# B&R Automation Studio project NAINV104C00R8L515F00 (part 33)

#### Act_Background_SendBoardDepartedLane3.st - Do Not Change!!!
```iecst
(** 2021-08-01 **)
ACTION Act_Background_SendBoardDepartedLane3: //Send after our machine send out "TransportFinished" message to downstream

	IF eStatus2 <> Error THEN
		IF tySServiceDescriptionRcv.tyData.tySupportedFeatures.bFeatureBoardTracking = TRUE AND p_tyParam.bFeatureBoardTracking AND bHandshakeDone THEN
			IF EDGEPOS(p_bDSHermesTransportFinished3) THEN

				fHermesAddOneMsgSend(ADR(a_eMsgSend) , ADR(udiMsgSendBffr) , HermesMsgTypeBoardDeparted3);

				tyBoardDeparted3.tyData.sMachineId     	        := p_sMcId;
			    tyBoardDeparted3.tyData.iDownstreamLaneId    	:= p_tyHermesConfiguration.a_tyDSParam[2].iLaneID;
			    tyBoardDeparted3.tyData.sDownstreamInterfaceId  := p_tyHermesConfiguration.a_tyDSParam[2].sDownstreamInterfaceId;
                tyBoardDeparted3.tyData.sMagazineId           	:= sMagazineId;
		    	tyBoardDeparted3.tyData.iSlotId     	        := iSlotId;
		    	tyBoardDeparted3.tyData.eBoadTransfer    	    := p_eBoardTransfer3;
	            tyBoardDeparted3.tyData.sBoardId     	        := p_tyDSBoardDeparted3.tyData.sBoardId;
		    	tyBoardDeparted3.tyData.sBoardIdCreatedBy     	:= p_tyDSBoardDeparted3.tyData.sBoardIdCreatedBy;
		    	tyBoardDeparted3.tyData.eFailedBoard			:= p_tyDSBoardDeparted3.tyData.eFailedBoard;
				tyBoardDeparted3.tyData.sProductTypeId			:= p_tyDSBoardDeparted3.tyData.sProductTypeId;
				tyBoardDeparted3.tyData.eFlippedBoard			:= p_tyDSBoardDeparted3.tyData.eFlippedBoard;
				tyBoardDeparted3.tyData.sTopBarcode				:= p_tyDSBoardDeparted3.tyData.sTopBarcode;
				tyBoardDeparted3.tyData.sBottomBarcode			:= p_tyDSBoardDeparted3.tyData.sBottomBarcode;
				tyBoardDeparted3.tyData.rLength					:= p_tyDSBoardDeparted3.tyData.rLength;
				tyBoardDeparted3.tyData.rWidth				    := p_tyDSBoardDeparted3.tyData.rWidth;
				tyBoardDeparted3.tyData.rThickness				:= p_tyDSBoardDeparted3.tyData.rThickness;
				tyBoardDeparted3.tyData.rConveyorSpeed		    := p_tyDSBoardDeparted3.tyData.rConveyorSpeed;
				tyBoardDeparted3.tyData.rTopClearanceHeight		:= p_tyDSBoardDeparted3.tyData.rTopClearanceHeight;
				tyBoardDeparted3.tyData.rBottomClearanceHeight	:= p_tyDSBoardDeparted3.tyData.rBottomClearanceHeight;
				tyBoardDeparted3.tyData.rWeight					:= p_tyDSBoardDeparted3.tyData.rWeight;
				tyBoardDeparted3.tyData.sWorkOrdedId            := p_tyDSBoardDeparted3.tyData.sWorkOrderId;
				tyBoardDeparted3.tyData.sBatchId                := p_tyDSBoardDeparted3.tyData.sBatchId;

			    tyBoardDeparted3.tyAvl.bMachineId				:= tyBoardDeparted3.tyData.sMachineId <> '';
		     	tyBoardDeparted3.tyAvl.bDownstreamLaneId		:= tyBoardDeparted3.tyData.iDownstreamLaneId <> 0;
		    	tyBoardDeparted3.tyAvl.bDownstreamInterfaceId	:= tyBoardDeparted3.tyData.sDownstreamInterfaceId <> '';
		    	tyBoardDeparted3.tyAvl.bMagazineId		    	:= tyBoardDeparted3.tyData.sMagazineId <> '';
		    	tyBoardDeparted3.tyAvl.bSlotId				    := tyBoardDeparted3.tyData.iSlotId <> 0;
		    	tyBoardDeparted3.tyAvl.bBoardTransfer		    := TRUE;
				tyBoardDeparted3.tyAvl.bBoardId					:= tyBoardDeparted3.tyData.sBoardId <> '';
				tyBoardDeparted3.tyAvl.bBoardIdCreatedBy		:= tyBoardDeparted3.tyData.sBoardIdCreatedBy <> '';
				tyBoardDeparted3.tyAvl.bFailedBoard				:= TRUE;
				tyBoardDeparted3.tyAvl.bProductTypeId		   	:= tyBoardDeparted3.tyData.sProductTypeId <> '';
				tyBoardDeparted3.tyAvl.bFlippedBoard			:= TRUE;
				tyBoardDeparted3.tyAvl.bTopBarcode			    := tyBoardDeparted3.tyData.sTopBarcode <> '';
				tyBoardDeparted3.tyAvl.bBottomBarcode		    := tyBoardDeparted3.tyData.sBottomBarcode <> '';
				tyBoardDeparted3.tyAvl.bLength				    := tyBoardDeparted3.tyData.rLength <> 0;
				tyBoardDeparted3.tyAvl.bWidth				    := (tyBoardDeparted3.tyData.rWidth <> 0);
				tyBoardDeparted3.tyAvl.bThickness			    := (tyBoardDeparted3.tyData.rThickness <> 0);
				tyBoardDeparted3.tyAvl.bConveyorSpeed		    := tyBoardDeparted3.tyData.rConveyorSpeed <> 0;
				tyBoardDeparted3.tyAvl.bTopClearanceHeight	    := (tyBoardDeparted3.tyData.rTopClearanceHeight <> 0);
				tyBoardDeparted3.tyAvl.bBottomClearanceHeight	:= (tyBoardDeparted3.tyData.rBottomClearanceHeight <> 0);
		    	tyBoardDeparted3.tyAvl.bWeight				    := tyBoardDeparted3.tyData.rWeight <> 0;
				tyBoardDeparted3.tyAvl.bWorkOrderId				:= tyBoardDeparted3.tyData.sWorkOrdedId <> '';
				tyBoardDeparted3.tyAvl.bBatchId			    	:= tyBoardDeparted3.tyData.sBatchId <> '';

			END_IF

		END_IF

	END_IF

END_ACTION
```

#### Act_Background_SendBoardDepartedLane4.st - Do Not Change!!!
```iecst
(** 2021-08-01 **)
ACTION Act_Background_SendBoardDepartedLane4: //Send after our machine send out "TransportFinished" message to downstream

	IF eStatus2 <> Error THEN
		IF tySServiceDescriptionRcv.tyData.tySupportedFeatures.bFeatureBoardTracking = TRUE AND p_tyParam.bFeatureBoardTracking AND bHandshakeDone THEN
			IF EDGEPOS(p_bDSHermesTransportFinished4) THEN

				fHermesAddOneMsgSend(ADR(a_eMsgSend) , ADR(udiMsgSendBffr) , HermesMsgTypeBoardDeparted4);

				tyBoardDeparted4.tyData.sMachineId     	        := p_sMcId;
			    tyBoardDeparted4.tyData.iDownstreamLaneId    	:= p_tyHermesConfiguration.a_tyDSParam[3].iLaneID;
			    tyBoardDeparted4.tyData.sDownstreamInterfaceId  := p_tyHermesConfiguration.a_tyDSParam[3].sDownstreamInterfaceId;
                tyBoardDeparted4.tyData.sMagazineId           	:= sMagazineId;
		    	tyBoardDeparted4.tyData.iSlotId     	        := iSlotId;
		    	tyBoardDeparted4.tyData.eBoadTransfer    	    := p_eBoardTransfer4;
	            tyBoardDeparted4.tyData.sBoardId     	        := p_tyDSBoardDeparted4.tyData.sBoardId;
		    	tyBoardDeparted4.tyData.sBoardIdCreatedBy     	:= p_tyDSBoardDeparted4.tyData.sBoardIdCreatedBy;
		    	tyBoardDeparted4.tyData.eFailedBoard			:= p_tyDSBoardDeparted4.tyData.eFailedBoard;
				tyBoardDeparted4.tyData.sProductTypeId			:= p_tyDSBoardDeparted4.tyData.sProductTypeId;
				tyBoardDeparted4.tyData.eFlippedBoard			:= p_tyDSBoardDeparted4.tyData.eFlippedBoard;
				tyBoardDeparted4.tyData.sTopBarcode				:= p_tyDSBoardDeparted4.tyData.sTopBarcode;
				tyBoardDeparted4.tyData.sBottomBarcode			:= p_tyDSBoardDeparted4.tyData.sBottomBarcode;
				tyBoardDeparted4.tyData.rLength					:= p_tyDSBoardDeparted4.tyData.rLength;
				tyBoardDeparted4.tyData.rWidth				    := p_tyDSBoardDeparted4.tyData.rWidth;
				tyBoardDeparted4.tyData.rThickness				:= p_tyDSBoardDeparted4.tyData.rThickness;
				tyBoardDeparted4.tyData.rConveyorSpeed		    := p_tyDSBoardDeparted4.tyData.rConveyorSpeed;
				tyBoardDeparted4.tyData.rTopClearanceHeight		:= p_tyDSBoardDeparted4.tyData.rTopClearanceHeight;
				tyBoardDeparted4.tyData.rBottomClearanceHeight	:= p_tyDSBoardDeparted4.tyData.rBottomClearanceHeight;
				tyBoardDeparted4.tyData.rWeight					:= p_tyDSBoardDeparted4.tyData.rWeight;
				tyBoardDeparted4.tyData.sWorkOrdedId            := p_tyDSBoardDeparted4.tyData.sWorkOrderId;
				tyBoardDeparted4.tyData.sBatchId                := p_tyDSBoardDeparted4.tyData.sBatchId;

			    tyBoardDeparted4.tyAvl.bMachineId				:= tyBoardDeparted4.tyData.sMachineId <> '';
		     	tyBoardDeparted4.tyAvl.bDownstreamLaneId		:= tyBoardDeparted4.tyData.iDownstreamLaneId <> 0;
		    	tyBoardDeparted4.tyAvl.bDownstreamInterfaceId	:= tyBoardDeparted4.tyData.sDownstreamInterfaceId <> '';
		    	tyBoardDeparted4.tyAvl.bMagazineId		    	:= tyBoardDeparted4.tyData.sMagazineId <> '';
		    	tyBoardDeparted4.tyAvl.bSlotId				    := tyBoardDeparted4.tyData.iSlotId <> 0;
		    	tyBoardDeparted4.tyAvl.bBoardTransfer		    := TRUE;
				tyBoardDeparted4.tyAvl.bBoardId					:= tyBoardDeparted4.tyData.sBoardId <> '';
				tyBoardDeparted4.tyAvl.bBoardIdCreatedBy		:= tyBoardDeparted4.tyData.sBoardIdCreatedBy <> '';
				tyBoardDeparted4.tyAvl.bFailedBoard				:= TRUE;
				tyBoardDeparted4.tyAvl.bProductTypeId		   	:= tyBoardDeparted4.tyData.sProductTypeId <> '';
				tyBoardDeparted4.tyAvl.bFlippedBoard			:= TRUE;
				tyBoardDeparted4.tyAvl.bTopBarcode			    := tyBoardDeparted4.tyData.sTopBarcode <> '';
				tyBoardDeparted4.tyAvl.bBottomBarcode		    := tyBoardDeparted4.tyData.sBottomBarcode <> '';
				tyBoardDeparted4.tyAvl.bLength				    := tyBoardDeparted4.tyData.rLength <> 0;
				tyBoardDeparted4.tyAvl.bWidth				    := (tyBoardDeparted4.tyData.rWidth <> 0);
				tyBoardDeparted4.tyAvl.bThickness			    := (tyBoardDeparted4.tyData.rThickness <> 0);
				tyBoardDeparted4.tyAvl.bConveyorSpeed		    := tyBoardDeparted4.tyData.rConveyorSpeed <> 0;
				tyBoardDeparted4.tyAvl.bTopClearanceHeight	    := (tyBoardDeparted4.tyData.rTopClearanceHeight <> 0);
				tyBoardDeparted4.tyAvl.bBottomClearanceHeight	:= (tyBoardDeparted4.tyData.rBottomClearanceHeight <> 0);
		    	tyBoardDeparted4.tyAvl.bWeight				    := tyBoardDeparted4.tyData.rWeight <> 0;
				tyBoardDeparted4.tyAvl.bWorkOrderId				:= tyBoardDeparted4.tyData.sWorkOrdedId <> '';
				tyBoardDeparted4.tyAvl.bBatchId			    	:= tyBoardDeparted4.tyData.sBatchId <> '';

			END_IF

		END_IF

	END_IF

END_ACTION
```

#### Act_Background_TCPSend.st - Do Not Change!!!
```iecst
(** 2021-08-01 **)
ACTION Act_Background_TCPSend:

	//Message Send (Generate XML Message)
	IF a_eMsgSend[0] <> HermesMsgTypeNA THEN

		IF a_eMsgSend[0] = HermesMsgTypeCheckAlive THEN
			fHermesFormCheckAlive(ADR(a_tyXMLTableDataSnd) , p_tyDTStructure , tyCheckAliveSnd);
			fTableConvertToXML(ADR(sSnd) , ADR(udiSndMsgLen) , SIZEOF(sSnd) , ADR(a_tyXMLTableDataSnd) , ADR(a_tyXMLTableDataSnd[0].sTitle) , ADR(a_tyXMLTableDataSnd[0].sValue) , ADR(a_tyXMLTableDataSnd[0].uiSize) , SIZEOF(a_tyXMLTableDataSnd[0]) , 12);

		ELSIF a_eMsgSend[0] = HermesMsgTypeCheckAlivePing THEN
			fHermesFormCheckAlive(ADR(a_tyXMLTableDataSnd) , p_tyDTStructure , tyCheckAlivePingSnd);
			fTableConvertToXML(ADR(sSnd) , ADR(udiSndMsgLen) , SIZEOF(sSnd) , ADR(a_tyXMLTableDataSnd) , ADR(a_tyXMLTableDataSnd[0].sTitle) , ADR(a_tyXMLTableDataSnd[0].sValue) , ADR(a_tyXMLTableDataSnd[0].uiSize) , SIZEOF(a_tyXMLTableDataSnd[0]) , 12);

		ELSIF a_eMsgSend[0] = HermesMsgTypeCheckAlivePong THEN
			fHermesFormCheckAlive(ADR(a_tyXMLTableDataSnd) , p_tyDTStructure , tyCheckAlivePongSnd);
			fTableConvertToXML(ADR(sSnd) , ADR(udiSndMsgLen) , SIZEOF(sSnd) , ADR(a_tyXMLTableDataSnd) , ADR(a_tyXMLTableDataSnd[0].sTitle) , ADR(a_tyXMLTableDataSnd[0].sValue) , ADR(a_tyXMLTableDataSnd[0].uiSize) , SIZEOF(a_tyXMLTableDataSnd[0]) , 12);

		ELSIF a_eMsgSend[0] = HermesMsgTypeSServiceDescription THEN
			fHermesFormSServiceDescription(ADR(a_tyXMLTableDataSnd) , p_tyDTStructure , tySServiceDescriptionSnd);
			fTableConvertToXML(ADR(sSnd) , ADR(udiSndMsgLen) , SIZEOF(sSnd) , ADR(a_tyXMLTableDataSnd) , ADR(a_tyXMLTableDataSnd[0].sTitle) , ADR(a_tyXMLTableDataSnd[0].sValue) , ADR(a_tyXMLTableDataSnd[0].uiSize) , SIZEOF(a_tyXMLTableDataSnd[0]) ,30);

		ELSIF a_eMsgSend[0] = HermesMsgTypeNotification THEN
			fHermesFormNotification(ADR(a_tyXMLTableDataSnd) , p_tyDTStructure , tyNotificationSnd);
			fTableConvertToXML(ADR(sSnd) , ADR(udiSndMsgLen) , SIZEOF(sSnd) , ADR(a_tyXMLTableDataSnd) , ADR(a_tyXMLTableDataSnd[0].sTitle) , ADR(a_tyXMLTableDataSnd[0].sValue) , ADR(a_tyXMLTableDataSnd[0].uiSize) , SIZEOF(a_tyXMLTableDataSnd[0]) , 14);

		ELSIF a_eMsgSend[0] = HermesMsgTypeBoardAvailable THEN
			eStatus1	:= Error;
			udiStatus1	:= 10125;	//Board Available Request To Send From Supervisory Hermes

		ELSIF a_eMsgSend[0] = HermesMsgTypeRevokeBoardAvl THEN
			eStatus1	:= Error;
			udiStatus1	:= 10122;	//Revoke Board Available Request To Send From Supervisory Hermes

		ELSIF a_eMsgSend[0] = HermesMsgTypeMachineReady THEN
			eStatus1	:= Error;
			udiStatus1	:= 10135;	//Machine Ready Request To Send From Supervisory Hermes

		ELSIF a_eMsgSend[0] = HermesMsgTypeRevokeMachineReady THEN
			eStatus1	:= Error;
			udiStatus1	:= 10136;	//Revoke Machine Ready Request To Send From Supervisory Hermes

		ELSIF a_eMsgSend[0] = HermesMsgTypeStartTransport THEN
			eStatus1	:= Error;
			udiStatus1	:= 10137;	//Start Transport Request To Send From Supervisory Hermes

		ELSIF a_eMsgSend[0] = HermesMsgTypeStopTransport THEN
			eStatus1	:= Error;
			udiStatus1	:= 10123;	//Stop Transport Request To Send From Supervisory Hermes

		ELSIF a_eMsgSend[0] = HermesMsgTypeTransportFinished THEN
			eStatus1	:= Error;
			udiStatus1	:= 10124;	//Transport Finished Request To Send From Supervisory Hermes

		ELSIF a_eMsgSend[0] = HermesMsgTypeSetConfiguration THEN
			eStatus1	:= Error;
			udiStatus1	:= 10138;	//Set Configuration Request To Send From Supervisory Hermes

		ELSIF a_eMsgSend[0] = HermesMsgTypeGetConfiguration THEN
			eStatus1	:= Error;
			udiStatus1	:= 10139;	//Get Configuration Request To Send From Supervisory Hermes

		ELSIF a_eMsgSend[0] = HermesMsgTypeCurrConfiguration THEN
			fHermesFormCurrentConfiguration(ADR(a_tyXMLTableDataSnd) , p_tyDTStructure , tyCurrentConfigurationSnd);
			fTableConvertToXML(ADR(sSnd) , ADR(udiSndMsgLen) , SIZEOF(sSnd) , ADR(a_tyXMLTableDataSnd) , ADR(a_tyXMLTableDataSnd[0].sTitle) , ADR(a_tyXMLTableDataSnd[0].sValue) , ADR(a_tyXMLTableDataSnd[0].uiSize) , SIZEOF(a_tyXMLTableDataSnd[0]) , 80);
			//10140

		ELSIF a_eMsgSend[0] = HermesMsgTypeBoardForecast THEN
			eStatus1	:= Error;
			udiStatus1	:= 10141;	//Board Forecast Request To Send From Supervisory Hermes

		ELSIF a_eMsgSend[0] = HermesMsgTypeQueryBoardInfo THEN
			eStatus1	:= Error;
			udiStatus1	:= 10142;	//Query Board Info Request To Send From Supervisory Hermes

		ELSIF a_eMsgSend[0] = HermesMsgTypeSendBoardInfo THEN
			eStatus1	:= Error;
			udiStatus1	:= 10159;	//Send Board Info Request To Send From Supervisory Hermes

	    ELSIF a_eMsgSend[0] = HermesMsgTypeQueryWorkOrderInfo THEN
	    	fHermesFormQueryWorkOrderInfo(ADR(a_tyXMLTableDataSnd) , p_tyDTStructure , tyQueryWorkOrderInfo);
		    fTableConvertToXML(ADR(sSnd) , ADR(udiSndMsgLen) , SIZEOF(sSnd) , ADR(a_tyXMLTableDataSnd) , ADR(a_tyXMLTableDataSnd[0].sTitle) , ADR(a_tyXMLTableDataSnd[0].sValue) , ADR(a_tyXMLTableDataSnd[0].uiSize) , SIZEOF(a_tyXMLTableDataSnd[0]) , 20);
			//10160

    	ELSIF a_eMsgSend[0] = HermesMsgTypeSendWorkOrderInfo THEN
	     	eStatus1	:= Error;
		    udiStatus1	:= 10161;	//Send Work Order Info Request To Send From Supervisory Hermes

	    ELSIF a_eMsgSend[0] = HermesMsgTypeBoardArrived1 THEN //Lane 1
		    fHermesFormBoardArrived(ADR(a_tyXMLTableDataSnd) , p_tyDTStructure , tyBoardArrived1);
		    fTableConvertToXML(ADR(sSnd) , ADR(udiSndMsgLen) , SIZEOF(sSnd) , ADR(a_tyXMLTableDataSnd) , ADR(a_tyXMLTableDataSnd[0].sTitle) , ADR(a_tyXMLTableDataSnd[0].sValue) , ADR(a_tyXMLTableDataSnd[0].uiSize) , SIZEOF(a_tyXMLTableDataSnd[0]) , 50);
			//10162

		ELSIF a_eMsgSend[0] = HermesMsgTypeBoardArrived2 THEN //Lane 2
			fHermesFormBoardArrived(ADR(a_tyXMLTableDataSnd) , p_tyDTStructure , tyBoardArrived2);
			fTableConvertToXML(ADR(sSnd) , ADR(udiSndMsgLen) , SIZEOF(sSnd) , ADR(a_tyXMLTableDataSnd) , ADR(a_tyXMLTableDataSnd[0].sTitle) , ADR(a_tyXMLTableDataSnd[0].sValue) , ADR(a_tyXMLTableDataSnd[0].uiSize) , SIZEOF(a_tyXMLTableDataSnd[0]) , 50);
			//10162

		ELSIF a_eMsgSend[0] = HermesMsgTypeBoardArrived3 THEN //Lane 3
			fHermesFormBoardArrived(ADR(a_tyXMLTableDataSnd) , p_tyDTStructure , tyBoardArrived3);
			fTableConvertToXML(ADR(sSnd) , ADR(udiSndMsgLen) , SIZEOF(sSnd) , ADR(a_tyXMLTableDataSnd) , ADR(a_tyXMLTableDataSnd[0].sTitle) , ADR(a_tyXMLTableDataSnd[0].sValue) , ADR(a_tyXMLTableDataSnd[0].uiSize) , SIZEOF(a_tyXMLTableDataSnd[0]) , 50);
			//10162

		ELSIF a_eMsgSend[0] = HermesMsgTypeBoardArrived4 THEN //Lane 4
			fHermesFormBoardArrived(ADR(a_tyXMLTableDataSnd) , p_tyDTStructure , tyBoardArrived4);
			fTableConvertToXML(ADR(sSnd) , ADR(udiSndMsgLen) , SIZEOF(sSnd) , ADR(a_tyXMLTableDataSnd) , ADR(a_tyXMLTableDataSnd[0].sTitle) , ADR(a_tyXMLTableDataSnd[0].sValue) , ADR(a_tyXMLTableDataSnd[0].uiSize) , SIZEOF(a_tyXMLTableDataSnd[0]) , 50);
			//10162

	    ELSIF a_eMsgSend[0] = HermesMsgTypeBoardDeparted1 THEN
	    	fHermesFormBoardDeparted(ADR(a_tyXMLTableDataSnd) , p_tyDTStructure , tyBoardDeparted1);
	    	fTableConvertToXML(ADR(sSnd) , ADR(udiSndMsgLen) , SIZEOF(sSnd) , ADR(a_tyXMLTableDataSnd) , ADR(a_tyXMLTableDataSnd[0].sTitle) , ADR(a_tyXMLTableDataSnd[0].sValue) , ADR(a_tyXMLTableDataSnd[0].uiSize) , SIZEOF(a_tyXMLTableDataSnd[0]) , 50);
			//10163

		ELSIF a_eMsgSend[0] = HermesMsgTypeBoardDeparted2 THEN
			fHermesFormBoardDeparted(ADR(a_tyXMLTableDataSnd) , p_tyDTStructure , tyBoardDeparted2);
			fTableConvertToXML(ADR(sSnd) , ADR(udiSndMsgLen) , SIZEOF(sSnd) , ADR(a_tyXMLTableDataSnd) , ADR(a_tyXMLTableDataSnd[0].sTitle) , ADR(a_tyXMLTableDataSnd[0].sValue) , ADR(a_tyXMLTableDataSnd[0].uiSize) , SIZEOF(a_tyXMLTableDataSnd[0]) , 50);
			//10163

		ELSIF a_eMsgSend[0] = HermesMsgTypeBoardDeparted3 THEN
			fHermesFormBoardDeparted(ADR(a_tyXMLTableDataSnd) , p_tyDTStructure , tyBoardDeparted3);
			fTableConvertToXML(ADR(sSnd) , ADR(udiSndMsgLen) , SIZEOF(sSnd) , ADR(a_tyXMLTableDataSnd) , ADR(a_tyXMLTableDataSnd[0].sTitle) , ADR(a_tyXMLTableDataSnd[0].sValue) , ADR(a_tyXMLTableDataSnd[0].uiSize) , SIZEOF(a_tyXMLTableDataSnd[0]) , 50);
			//10163

		ELSIF a_eMsgSend[0] = HermesMsgTypeBoardDeparted4 THEN
			fHermesFormBoardDeparted(ADR(a_tyXMLTableDataSnd) , p_tyDTStructure , tyBoardDeparted4);
			fTableConvertToXML(ADR(sSnd) , ADR(udiSndMsgLen) , SIZEOF(sSnd) , ADR(a_tyXMLTableDataSnd) , ADR(a_tyXMLTableDataSnd[0].sTitle) , ADR(a_tyXMLTableDataSnd[0].sValue) , ADR(a_tyXMLTableDataSnd[0].uiSize) , SIZEOF(a_tyXMLTableDataSnd[0]) , 50);
			//10163

		ELSIF a_eMsgSend[0] = HermesMsgTypeReplyWorkOrderInfo THEN
			fHermesFormReplyWorkOrderInfo(ADR(a_tyXMLTableDataSnd) , p_tyDTStructure , tyReplyWorkOrderInfo);
			fTableConvertToXML(ADR(sSnd) , ADR(udiSndMsgLen) , SIZEOF(sSnd) , ADR(a_tyXMLTableDataSnd) , ADR(a_tyXMLTableDataSnd[0].sTitle) , ADR(a_tyXMLTableDataSnd[0].sValue) , ADR(a_tyXMLTableDataSnd[0].uiSize) , SIZEOF(a_tyXMLTableDataSnd[0]) , 20);
			//10164    //ADD

		END_IF

		//Message Send
		IF p_bInternalUse = FALSE THEN
			fbSend.udiTCPIdent	:= udiClntIdent;
			fbSend.udiSndSize	:= udiSndMsgLen;
			fbSend(bEn := TRUE);
		ELSE
			sInternalSnd	:= sSnd;
		END_IF

		IF (fbSend.udiStatus = 0) OR (p_bInternalUse = TRUE) THEN

			fLogDTConvert(ADR(sDT) , p_dtCurrDT);
			memset(ADR(a_sLogList[udiLogCntr]) , 0 , SIZEOF(a_sLogList[udiLogCntr]));
			memcpy(ADR(a_sLogList[udiLogCntr]) + LEN(a_sLogList[udiLogCntr]) , ADR(sDT) , LEN(sDT));
			memcpy(ADR(a_sLogList[udiLogCntr]) + LEN(a_sLogList[udiLogCntr]) , ADR('$r$n') , LEN('$r$n'));
			memcpy(ADR(a_sLogList[udiLogCntr]) + LEN(a_sLogList[udiLogCntr]) , ADR('SND_TO_SVY$r$n') , LEN('SND_TO_SVY$r$n'));
			memcpy(ADR(a_sLogList[udiLogCntr]) + LEN(a_sLogList[udiLogCntr]) , ADR(sSnd) , LEN(sSnd));
			memcpy(ADR(a_sLogList[udiLogCntr]) + LEN(a_sLogList[udiLogCntr]) , ADR('$r$n$r$n') , LEN('$r$n$r$n'));

			udiLogCntr	:= udiLogCntr + 1;
			IF udiLogCntr = 11 THEN
				udiLogCntr	:= 1;
			END_IF

			Act_Background_NotificationSnd;
			fHermesRmvOneMsgSend(ADR(a_eMsgSend) , ADR(udiMsgSendBffr));

			fbSend(bEn := FALSE);

		ELSIF (fbSend.udiStatus = 2321) AND (p_bInternalUse = FALSE) THEN
			bRstConnection	:= TRUE;

		ELSIF (fbSend.udiStatus < 65534) AND (p_bInternalUse = FALSE) THEN
			eStatus1	:= Error;

			IF fbSend.udiStatus = 2300 THEN
				udiStatus1	:= 10143;	//Invalid Ident While Sending Data
			ELSIF fbSend.udiStatus = 2320 THEN
				udiStatus1	:= 10144;	//TCP Retry Send Data Error While Sending Data
			ELSIF fbSend.udiStatus = 2322 THEN
				udiStatus1	:= 10145;	//TCP Send Data Error
			ELSE
				udiStatus1	:= fbSend.udiStatus;
			END_IF

	    END_IF
	END_IF

END_ACTION
```

#### Act_Background_TCPCloseSvr.st - Do Not Change!!!
```iecst
(** 2021-08-01 **)
ACTION Act_Background_TCPCloseSvr:

	//Close Server Connection
	IF p_bInternalUse = FALSE THEN
		fbCloseSvr.udiTCPIdent	:= udiSvrIdent;
		fbCloseSvr(bEn := TRUE);

		IF fbCloseSvr.udiStatus = 0 THEN
			udiSvrIdent		:= 0;
			fbCloseSvr(bEn := FALSE);

		ELSIF fbCloseSvr.udiStatus < 65534 THEN
			udiSvrIdent		:= 0;
			eStatus1		:= Error;

			IF fbCloseSvr.udiStatus = 2300 THEN
				udiStatus1	:= 10146;	//Invalid Ident While Closing TCP
			ELSIF fbCloseSvr.udiStatus = 2310 THEN
				udiStatus1	:= 10147;	//Closing TCP Error
			ELSE
				udiStatus1	:= fbCloseSvr.udiStatus;
			END_IF

		END_IF

	ELSE
		udiSvrIdent	:= 0;

	END_IF

END_ACTION
```

#### Act_Background_TCPCloseClnt.st - Do Not Change!!!
```iecst
(** 2021-08-01 **)
ACTION Act_Background_TCPCloseClnt:

	//Close Server Connection
	IF p_bInternalUse = FALSE THEN
		fbCloseClnt.udiTCPIdent	:= udiClntIdent;
		fbCloseClnt(bEn := TRUE);

		IF fbCloseClnt.udiStatus = 0 THEN
			udiClntIdent	:= 0;
			fbCloseClnt(bEn := FALSE);

		ELSIF fbCloseClnt.udiStatus < 65534 THEN
			udiClntIdent	:= 0;
			eStatus1		:= Error;

			IF fbCloseClnt.udiStatus = 2300 THEN
				udiStatus1	:= 10154;	//Invalid Ident While Closing TCP
			ELSIF fbCloseClnt.udiStatus = 2310 THEN
				udiStatus1	:= 10155;	//Closing TCP Error
			ELSE
				udiStatus1	:= fbCloseClnt.udiStatus;
			END_IF

		END_IF

	ELSE
		udiClntIdent	:= 0;

	END_IF

END_ACTION
```

#### Act_Background_Log.st - Do Not Change!!!
```iecst
(** 2021-08-01 **)
ACTION Act_Background_Log:

	IF eStatus3 <> Error THEN

		IF udiWriteLogCntr <> udiLogCntr THEN

			CASE iWriteLogStep OF

				0:
					dtCurrDTTemp			:= p_dtCurrDT;
					fbFileAppend1.sFile		:= DT_TO_STRING(dtCurrDTTemp);
					fbFileAppend1.sFile		:= MID(fbFileAppend1.sFile , 10 , 4);
					fbFileAppend1.sFile		:= CONCAT('_' , fbFileAppend1.sFile);
					fbFileAppend1.sFile		:= CONCAT(p_sProgNm , fbFileAppend1.sFile);
					fbFileAppend1.sFile		:= CONCAT(fbFileAppend1.sFile , '.dat');

					fbFileAppend1.p_Src		:= ADR(a_sLogList[udiWriteLogCntr]);
					fbFileAppend1.udiLen	:= LEN(a_sLogList[udiWriteLogCntr]);

					iWriteLogStep	:= 1;

				1:
					fbFileAppend1(bEn := TRUE);
					IF fbFileAppend1.udiStatus = 0 THEN
						fbFileAppend1(bEn := FALSE);

						udiWriteLogCntr	:= udiWriteLogCntr + 1;
						IF udiWriteLogCntr = 11 THEN
							udiWriteLogCntr	:= 1;
						END_IF

						iWriteLogStep	:= 0;

					ELSIF fbFileAppend1.udiStatus < 65534 THEN
						eStatus3	:= Error;

						IF fbFileAppend1.udiStatus = 1900 THEN
							udiStatus3	:= 10148;	//File Open Error While Writing Log
						ELSIF fbFileAppend1.udiStatus = 1901 THEN
							udiStatus3	:= 10149;	//File Create Error While Writing Log
						ELSIF fbFileAppend1.udiStatus = 1913 THEN
							udiStatus3	:= 10150;	//Get File Info Error While Writing Log
						ELSIF fbFileAppend1.udiStatus = 1903 THEN
							udiStatus3	:= 10151;	//File Write Error While Writing Log
						ELSIF fbFileAppend1.udiStatus = 1904 THEN
							udiStatus3	:= 10152;	//File Close Error While Writing Log
						ELSIF fbFileAppend1.udiStatus = 1914 THEN
							udiStatus3	:= 10153;	//Directory Does Not Exist While Writing Log
						ELSE
							udiStatus3	:= fbFileAppend1.udiStatus;
						END_IF

						iWriteLogStep	:= 0;
					END_IF

			END_CASE

		END_IF

	END_IF

END_ACTION
```

#### Act_Background_Err.st - Do Not Change!!!
```iecst
(** 2021-08-01 **)
ACTION Act_Background_Err:

END_ACTION
```

#### Act_Main_Disable.st - Do Not Change!!!
```iecst
(** 2021-08-01 **)
ACTION Act_Main_Disable:

	bConnected		:= FALSE;
	bHandshakeDone	:= FALSE;

END_ACTION
```

#### Act_CombineErr.st - Do Not Change!!!
```iecst
(** 2021-08-01 **)
ACTION Act_CombineErr:

	//Combine Error
	IF eStatus = Error OR eStatus1 = Error OR eStatus2 = Error OR eStatus3 = Error THEN
		eMainStatus	:= Error;
	ELSE
		eMainStatus	:= eStatus;
	END_IF

END_ACTION
```

#### Act_Alarm.st - Do Not Change!!!
```iecst
(** 2021-08-01 **)
ACTION Act_Alarm: //General

	//Error
	IF EDGEPOS(eStatus = Error) THEN

		tyAlmData.sProgNm		:= p_sProgNm;
		tyAlmData.udiCode		:= udiStatus;
		tyAlmData.eSeverity		:= AlmSeverityError;
		tyAlmData.udiRunTime	:= tyAlmData.udiRunTime + 1;
		tyAlmData.bAlm			:= TRUE;
		tyAlmData.udiModuleNum  := udiModuleNum;
		g_sSvyHermesProgNm		:= p_sProgNm;
		//Get Error Message
		IF tyAlmData.udiCode < 10000 OR tyAlmData.udiCode > 10199 THEN
			tyAlmData.sAlmMsg	:= 'Unknown';
			tyAlmData.sRcyMsg	:= 'Unknown';
		ELSE
			tyAlmData.sAlmMsg	:= a_tyAlmText[tyAlmData.udiCode].sAlmText;
			tyAlmData.sRcyMsg	:= a_tyAlmText[tyAlmData.udiCode].sRcyText;
		END_IF

		sStatTxt	:= tyAlmData.sAlmMsg;

	ELSIF bRstErr AND (tyAlmData.udiCode <> 0) THEN

		tyAlmData.udiCode	:= 0;
		tyAlmData.eSeverity	:= AlmSeverityNA;
		tyAlmData.sAlmMsg	:= '';
		tyAlmData.sRcyMsg	:= '';
		tyAlmData1.bAlm			:= FALSE;
		sStatTxt	:= a_sStatText[eStat];

	END_IF

END_ACTION
```

#### Act_Alarm1.st - Do Not Change!!!
```iecst
(** 2021-08-01 **)
ACTION Act_Alarm1:

	//Error
	IF EDGEPOS(eStatus1 = Error) THEN

		tyAlmData1.sProgNm		:= p_sProgNm;
		tyAlmData1.udiCode		:= udiStatus1;
		tyAlmData1.eSeverity	:= AlmSeverityError;
		tyAlmData1.udiRunTime	:= tyAlmData1.udiRunTime + 1;
		tyAlmData1.bAlm			:= TRUE;
		tyAlmData1.udiModuleNum := udiModuleNum;
		g_sSvyHermesProgNm		:= p_sProgNm;
		//Get Error Message
		IF tyAlmData1.udiCode < 10000 OR tyAlmData1.udiCode > 10199 THEN
			tyAlmData1.sAlmMsg	:= 'Unknown';
			tyAlmData1.sRcyMsg	:= 'Unknown';
		ELSE
			tyAlmData1.sAlmMsg	:= a_tyAlmText[tyAlmData1.udiCode].sAlmText;
			tyAlmData1.sRcyMsg	:= a_tyAlmText[tyAlmData1.udiCode].sRcyText;
		END_IF

		sStatTxt	:= tyAlmData1.sAlmMsg;

	ELSIF bRstErr AND (tyAlmData1.udiCode <> 0) THEN

		tyAlmData1.udiCode		:= 0;
		tyAlmData1.eSeverity	:= AlmSeverityNA;
		tyAlmData1.sAlmMsg		:= '';
		tyAlmData1.sRcyMsg		:= '';
		tyAlmData1.bAlm			:= FALSE;
		sStatTxt	:= a_sStatText[eStat];

	END_IF

END_ACTION
```

#### Act_Alarm2.st - Do Not Change!!!
```iecst
(** 2021-08-01 **)
ACTION Act_Alarm2:

	//Error
	IF EDGEPOS(eStatus2 = Error) THEN

		tyAlmData2.sProgNm		:= p_sProgNm;
		tyAlmData2.udiCode		:= udiStatus2;
		tyAlmData2.eSeverity	:= AlmSeverityError;
		tyAlmData2.udiRunTime	:= tyAlmData2.udiRunTime + 1;
		tyAlmData2.bAlm			:= TRUE;
		tyAlmData2.udiModuleNum := udiModuleNum;
		g_sSvyHermesProgNm		:= p_sProgNm;
		//Get Error Message
		IF tyAlmData2.udiCode < 10000 OR tyAlmData2.udiCode > 10199 THEN
			tyAlmData2.sAlmMsg	:= 'Unknown';
			tyAlmData2.sRcyMsg	:= 'Unknown';
		ELSE
			tyAlmData2.sAlmMsg	:= a_tyAlmText[tyAlmData2.udiCode].sAlmText;
			tyAlmData2.sRcyMsg	:= a_tyAlmText[tyAlmData2.udiCode].sRcyText;
		END_IF

		sStatTxt	:= tyAlmData2.sAlmMsg;

	ELSIF bRstErr AND (tyAlmData2.udiCode <> 0) THEN

		tyAlmData2.udiCode		:= 0;
		tyAlmData2.eSeverity	:= AlmSeverityNA;
		tyAlmData2.sAlmMsg		:= '';
		tyAlmData2.sRcyMsg		:= '';
		tyAlmData2.bAlm			:= FALSE;
		sStatTxt	:= a_sStatText[eStat];

	END_IF

END_ACTION
```

#### Act_Alarm3.st - Do Not Change!!!
```iecst
(** 2021-08-01 **)
ACTION Act_Alarm3: //fbFileAppend1 Error

	//Error
	IF EDGEPOS(eStatus3 = Error) THEN

		tyAlmData3.sProgNm		:= p_sProgNm;
		tyAlmData3.udiCode		:= udiStatus3;
		tyAlmData3.eSeverity	:= AlmSeverityError;
		tyAlmData3.udiRunTime	:= tyAlmData3.udiRunTime + 1;
		tyAlmData3.bAlm			:= TRUE;
		tyAlmData3.udiModuleNum := udiModuleNum;
		g_sSvyHermesProgNm		:= p_sProgNm;
		//Get Error Message
		IF tyAlmData3.udiCode < 10000 OR tyAlmData3.udiCode > 10199 THEN
			tyAlmData3.sAlmMsg	:= 'Unknown';
			tyAlmData3.sRcyMsg	:= 'Unknown';
		ELSE
			tyAlmData3.sAlmMsg	:= a_tyAlmText[tyAlmData3.udiCode].sAlmText;
			tyAlmData3.sRcyMsg	:= a_tyAlmText[tyAlmData3.udiCode].sRcyText;
		END_IF

		sStatTxt	:= tyAlmData3.sAlmMsg;

	ELSIF bRstErr AND (tyAlmData3.udiCode <> 0) THEN

		tyAlmData3.udiCode		:= 0;
		tyAlmData3.eSeverity	:= AlmSeverityNA;
		tyAlmData3.sAlmMsg		:= '';
		tyAlmData3.sRcyMsg		:= '';
		tyAlmData3.bAlm			:= FALSE;
		sStatTxt	:= a_sStatText[eStat];

	END_IF

END_ACTION
```

#### Act_Alarm4.st - Do Not Change!!!
```iecst
(** 2021-08-01 **)
ACTION Act_Alarm4: //Not Connected Warning

	//Warning
	IF ((bConnected = FALSE) AND (p_bSvyEn)) THEN

		tyAlmData4.sProgNm		:= p_sProgNm;
		tyAlmData4.udiCode		:= udiStatus4;
		tyAlmData4.eSeverity	:= AlmSeverityWarning;
		tyAlmData4.udiRunTime	:= tyAlmData4.udiRunTime + 1;
		//tyUIAlmData.bWarning[6663] := TRUE;			// (05042023)Debug Alarm Test
		tyAlmData4.bWarning			:= TRUE;
		tyAlmData4.udiModuleNum := udiModuleNum;
		g_sSvyHermesProgNm		:= p_sProgNm;
		//Get Warning Message
		IF tyAlmData4.udiCode < 10000 OR tyAlmData4.udiCode > 10199 THEN
			tyAlmData4.sAlmMsg	:= 'Unknown';
			tyAlmData4.sRcyMsg	:= 'Unknown';
		ELSE
			tyAlmData4.sAlmMsg	:= a_tyAlmText[tyAlmData4.udiCode].sAlmText;
			tyAlmData4.sRcyMsg	:= a_tyAlmText[tyAlmData4.udiCode].sRcyText;
		END_IF

		sStatTxt	:= tyAlmData4.sAlmMsg;

	ELSIF (bConnected AND (tyAlmData4.udiCode <> 0)) OR (p_bSvyEn = FALSE) THEN

		tyAlmData4.udiCode		:= 0;
		tyAlmData4.eSeverity	:= AlmSeverityNA;
		tyAlmData4.sAlmMsg		:= '';
		tyAlmData4.sRcyMsg		:= '';
		//tyUIAlmData.bWarning[6663] := FALSE;		// (05042023)Debug Alarm Test
		tyAlmData4.bWarning			:= FALSE;
		sStatTxt	:= a_sStatText[eStat];

	END_IF

END_ACTION
```

#### InputRef.var - Do Not Change!!!
```iecst
(*2021-08-01*)
(**)
(*Configuration*)
VAR
	p_tyParam : REFERENCE TO tyHermesSvyParam;
	p_sIPAddr : REFERENCE TO STRING[15];
	pa_usiMacAddr : REFERENCE TO ARRAY[0..5] OF USINT;
	p_tyDTStructure : REFERENCE TO DTStructure;
	p_dtCurrDT : REFERENCE TO DATE_AND_TIME;
	p_sMcId : REFERENCE TO STRING[80];
END_VAR
(**)
(*General*)
VAR
	p_eAct : REFERENCE TO eHermesAction;
	p_udiRstErr : REFERENCE TO UDINT;
	p_bPrep : REFERENCE TO BOOL;
	p_bEn : REFERENCE TO BOOL;
	p_bDis : REFERENCE TO BOOL;
END_VAR
(**)
(*Input*)
VAR
	p_sRecipeNm : REFERENCE TO STRING[254];
	p_sMagazineId : REFERENCE TO STRING[80];
	p_iSlotId : REFERENCE TO INT;
	p_eBoardTransfer1 : REFERENCE TO eHermesBoardTransfer;
	p_eBoardTransfer2 : REFERENCE TO eHermesBoardTransfer;
	p_eBoardTransfer3 : REFERENCE TO eHermesBoardTransfer;
	p_eBoardTransfer4 : REFERENCE TO eHermesBoardTransfer;
	p_sBarcode : REFERENCE TO STRING[254];
	p_sVersion : REFERENCE TO STRING[7];
	p_udiSndBffrSize : REFERENCE TO UDINT;
	p_udiRcvBffrSize : REFERENCE TO UDINT;
	p_udiAliveIdleTimeInSec : REFERENCE TO UDINT;
	p_tConnTimeOut : REFERENCE TO TIME;
	p_diTransferInTO : REFERENCE TO DINT;
	p_bNewBrdAvlLastZone : REFERENCE TO BOOL;
	p_bOpsRun : REFERENCE TO BOOL;
	p_udiFileKeepDay : REFERENCE TO UDINT;
	p_sConfigFileName : REFERENCE TO STRING[80];
	p_sProgNm : REFERENCE TO STRING[15];
	p_bNtSettingsLoadDone : REFERENCE TO BOOL;
	p_bSvyPrep : REFERENCE TO BOOL;
	p_bSvyEn : REFERENCE TO BOOL;
	p_bQueryWorkOrderInfo : REFERENCE TO BOOL;
	p_bReinsertBrd : REFERENCE TO BOOL;
	p_bInsertBoard : REFERENCE TO BOOL;
	p_tyHermesConfiguration : REFERENCE TO tyHermesConfiguration;
	p_bUSHermesStopTransport1 : REFERENCE TO BOOL;
	p_bUSHermesStopTransport2 : REFERENCE TO BOOL;
	p_bUSHermesStopTransport3 : REFERENCE TO BOOL;
	p_bUSHermesStopTransport4 : REFERENCE TO BOOL;
	p_tyUSBoardArrived1 : REFERENCE TO tyHermesBoardAvailable;
	p_tyUSBoardArrived2 : REFERENCE TO tyHermesBoardAvailable;
	p_tyUSBoardArrived3 : REFERENCE TO tyHermesBoardAvailable;
	p_tyUSBoardArrived4 : REFERENCE TO tyHermesBoardAvailable;
	p_bDSHermesTransportFinished1 : REFERENCE TO BOOL;
	p_bDSHermesTransportFinished2 : REFERENCE TO BOOL;
	p_bDSHermesTransportFinished3 : REFERENCE TO BOOL;
	p_bDSHermesTransportFinished4 : REFERENCE TO BOOL;
	p_tyDSBoardDeparted1 : REFERENCE TO tyHermesBoardAvailable;
	p_tyDSBoardDeparted2 : REFERENCE TO tyHermesBoardAvailable;
	p_tyDSBoardDeparted3 : REFERENCE TO tyHermesBoardAvailable;
	p_tyDSBoardDeparted4 : REFERENCE TO tyHermesBoardAvailable;
	p_udiRetainDataAddr : REFERENCE TO UDINT;
	p_udiRetainDataLen : REFERENCE TO UDINT;
	p_sInfoMsg : REFERENCE TO STRING[200];
	p_sInfoMsg1 : REFERENCE TO STRING[200];
	p_sInfoMsg2 : REFERENCE TO STRING[200];
	p_sInfoMsg3 : REFERENCE TO STRING[200];
	p_sInfoMsg4 : REFERENCE TO STRING[200];
	p_sInfoMsg5 : REFERENCE TO STRING[200];
	p_sInfoMsg6 : REFERENCE TO STRING[200];
	p_eMcParamStatus : REFERENCE TO eFBStatus;
	p_eMcParamStat : REFERENCE TO eMcParamAction;
	p_eHermesStatus : REFERENCE TO eFBStatus;
	p_eHermesStat : REFERENCE TO eHermesAction;
	p_bAllZonesEmpty : REFERENCE TO BOOL;
	p_bDeleteWorkOrder : REFERENCE TO BOOL;
	p_bFirstMcIntheLine : REFERENCE TO BOOL;
	p_sRetainFileName : REFERENCE TO STRING[80];
	p_sInternalRcv : REFERENCE TO STRING[65535];
	p_bInternalUse : REFERENCE TO BOOL;
	p_bHermesSvyQueryBoardInfo : REFERENCE TO BOOL;
	p_bHermesReinsertBoard : REFERENCE TO BOOL;
	p_bAcceptCondition : REFERENCE TO BOOL;
	p_bConvRgtSen : REFERENCE TO BOOL;
	p_bConvLftSen : REFERENCE TO BOOL;
	p_bAWWidthPosDiff : REFERENCE TO BOOL;
	p_bOpsGConvStepDSTmr : REFERENCE TO BOOL;
	p_bOpsGConvStepDSCommTmr : REFERENCE TO BOOL;
	p_bOpsGConvStepEntBrd : REFERENCE TO BOOL;
	p_tyProdRcpCurrRcp : REFERENCE TO tyProdRcpParam;
	p_tyMcParamCurr : REFERENCE TO tyMcParam;
	p_tyNtParamCurr : REFERENCE TO tyNtParam;
	p_eLinkMcParamDSCommMod : REFERENCE TO eMcSetCommMod;
END_VAR
```

#### Local.var - Do Not Change!!!
```iecst
(*2021-08-01*)
(**)
(*Local Action, State & Status*)
VAR
	eAct : eHermesAction := HermesActIdle;
	eStat : eHermesAction := HermesActIdle;
	eHermesAct : eHermesAction;
	eMcParamAct : eMcParamAction;
	eMainStatus : eFBStatus := Idle;
	eStatus : eFBStatus := Idle;
	eStatus1 : eFBStatus := Idle;
	eStatus2 : eFBStatus := Idle;
	eStatus3 : eFBStatus := Idle;
	udiStatus : UDINT := 0;
	udiStatus1 : UDINT := 0;
	udiStatus2 : UDINT := 0;
	udiStatus3 : UDINT := 0;
	udiStatus4 : UDINT := 0;
	sStatTxt : STRING[200] := '';
	a_sStatText : ARRAY[0..50] OF STRING[200] := ['Idling','Background Starting Operations','Background Stopping Operations','Deleting Old Log File','Creating Directory','Writing Retain File','Reading Retain File','Saving Configuration',43('')];
END_VAR
(**)
(*Local Alarm*)
VAR
	tyAlmData : tyAlmDat;
	tyAlmData1 : tyAlmDat;
	tyAlmData2 : tyAlmDat;
	tyAlmData3 : tyAlmDat;
	tyAlmData4 : tyAlmDat;
	tyInfoData : tyAlmDat;
	tyInfoData1 : tyAlmDat;
	tyInfoData2 : tyAlmDat;
	tyInfoData3 : tyAlmDat;
	tyInfoData4 : tyAlmDat;
	tyInfoData5 : tyAlmDat;
	tyInfoData6 : tyAlmDat;
	a_tyAlmText : ARRAY[10000..10199] OF tyAlmTxt := [(sAlmText:='Invalid Ident While Creating Server',sRcyText:='Problem Occurred In The TCP/IP Connection. Check The Connection And Try To Reconnect.'),(sAlmText:='Setting Keep Alive Interval Time Error While Creating Server',sRcyText:='Unable To Establish Connection Between Machine. Check For Setting And Resume Operation.'),(sAlmText:='Setting Keep Alive Idle Time Error While Creating Server',sRcyText:='Unable To Establish Connection Between Machine. Check For Setting And Resume Operation.'),(sAlmText:='Setting Keep Alive Count Error While Creating Server',sRcyText:='Unable To Establish Connection Between Machine. Check For Setting And Resume Operation.'),(sAlmText:='Setting Keep Alive Error While Creating Server',sRcyText:='Unable To Establish Connection Between Machine. Check For Setting And Resume Operation.'),(sAlmText:='Setting Receive Buffer Error While Creating Server',sRcyText:='Unable To Establish Connection Between Machine. Check For Setting And Resume Operation.'),(sAlmText:='Setting Send Buffer Error While Creating Server',sRcyText:='Unable To Establish Connection Between Machine. Check For Setting And Resume Operation.'),(sAlmText:='Setting No Waiting Error While Creating Server',sRcyText:='Unable To Establish Connection Between Machine. Check For Setting And Resume Operation.'),(sAlmText:='TCP Open Port Error While Creating Server',sRcyText:='Problem Occurred In The TCP/IP Connection. Check The Connection And Try To Reconnect.'),(sAlmText:='Closing TCP Error While Creating Server',sRcyText:='Problem Occurred In The TCP/IP Connection. Check The Connection And Try To Reconnect.'),(sAlmText:='Invalid Ident While Listening Client',sRcyText:='There Was A Problem Connecting To The Server. The Server May Not Exist or It is Unavailable At This Time. Check The Connection and Try Again.'),0,(sAlmText:='Supervisory Hermes Connection Lost',sRcyText:='There Was A Problem Connecting To The Server. The Server May Not Exist or It is Unavailable At This Time. Check The Connection and Try Again.'),0,(sAlmText:='Invalid Ident While Receiving Data',sRcyText:='Problem Occurred In The TCP/IP Connection. Check The Connection And Try To Reconnect.'),(sAlmText:='TCP Receive Data Error While Receiving Data',sRcyText:='Problem Occurred In The TCP/IP Connection. Check The Connection And Try To Reconnect.'),(sAlmText:='Receive SetConfiguration While Supervisory In Not Connected State',sRcyText:='Receive Illegal Message.'),(sAlmText:='Receive GetConfiguration While Supervisory In Not Connected State',sRcyText:='Receive Illegal Message.'),(sAlmText:='Receive CurrConfiguration While Supervisory In Not Connected State',sRcyText:='Receive Illegal Message.'),(sAlmText:='Receive SendWorkOrderInfo While Supervisory In Not Connected State',sRcyText:='Receive Illegal Message.'),(sAlmText:='Receive QueryWorkOrderInfo While Supervisory In Not Connected State',sRcyText:='Receive Illegal Message.'),(sAlmText:='Receive BoardArrived While Supervisory In Not Connected State',sRcyText:='Receive Illegal Message.'),(sAlmText:='Receive BoardDeparted While Supervisory In Not Connected State',sRcyText:='Receive Illegal Message.'),2(0),(sAlmText:='Receive BoardAvailable While Downstream In Service Description State',sRcyText:='Receive Illegal Message.'),(sAlmText:='Receive RevokeBoardAvailable While Downstream In Service Description State',sRcyText:='Receive Illegal Message.'),(sAlmText:='Receive ServiceDescription While Supervisory In Service Description State',sRcyText:='Receive Illegal Message.'),(sAlmText:='Receive SetConfiguration While Supervisory In Service Description State',sRcyText:='Receive Illegal Message.'),(sAlmText:='Receive GetConfiguration While Supervisory In Service Description State',sRcyText:='Receive Illegal Message.'),(sAlmText:='Receive CurrConfiguration While Supervisory In Service Description State',sRcyText:='Receive Illegal Message.'),(sAlmText:='Receive SendWorkOrderInfo While Supervisory In Service Description State',sRcyText:='Receive Illegal Message.'),(sAlmText:='Receive QueryWorkOrderInfo While Supervisory In Service Description State',sRcyText:='Receive Illegal Message.'),(sAlmText:='Receive BoardArrived While Supervisory In Service Description State',sRcyText:='Receive Illegal Message.'),(sAlmText:='Receive BoardDeparted While Supervisory In Service Description State',sRcyText:='Receive Illegal Message.'),4(0),(sAlmText:='Receive ServiceDescription While Supervisory In Connected State',sRcyText:='Receive Illegal Message.'),(sAlmText:='Receive CurrConfiguration While Supervisory In Connected State',sRcyText:='Receive Illegal Message.'),(sAlmText:='Receive QueryWorkOrderInfo While Supervisory In Connected State',sRcyText:='Receive Illegal Message.'),(sAlmText:='Receive BoardArrived While Supervisory In Connected State',sRcyText:='Receive Illegal Message.'),(sAlmText:='Receive BoardDeparted While Supervisory In Connected State',sRcyText:='Receive Illegal Message.'),43(0),(sAlmText:='SystemId Missing While Checking Service Description',sRcyText:='Missing Input Value For SystemId. Fill Up The Value And Resend.'),(sAlmText:='Version Missing While Checking Service Description',sRcyText:='Missing Input Value For Version. Fill Up The Value And Resend.'),(sAlmText:='SupportedFeatures Missing While Checking Service Description',sRcyText:='Missing Input Value For SupportedFeatures. Fill Up The Value And Resend.'),2(0),(sAlmText:='NotificationCode Out Of Range While Checking Notification',sRcyText:='NotificationCode Does Not Fall Within The Expected Range.'),(sAlmText:='NotificationCode Missing While Checking Notification',sRcyText:='Missing Input Value For NotificationCode. Fill Up The Value And Resend.'),(sAlmText:='Severity Missing While Checking Notification',sRcyText:='Missing Input Value For Severity. Fill Up The Value And Resend.'),(sAlmText:='Description Missing While Checking Notification',sRcyText:='Missing Input Value For Description. Fill Up The Value And Resend.'),10(0),(sAlmText:='Supervisory Service Description Interchange Time Out',sRcyText:='Timeout Expired Before Operation Completed. Reset And Resume Operation.'),4(0),(sAlmText:='Get Directory Info Error While Deleting Old Log',sRcyText:='An Error Was Encountered While Getting Directory Info. Please Contact Nutek For A Possible Solution.'),(sAlmText:='Directory Read Error While Deleting Old Log',sRcyText:='An Error Was Encountered While Reading Directory. Please Contact Nutek For A Possible Solution.'),(sAlmText:='File Delete Error While Deleting Old Log',sRcyText:='An Error Was Encountered While Trying To Delete File. Please Contact Nutek For A Possible Solution.'),(sAlmText:='File Open Error While Reading Retain File',sRcyText:='An Error Was Encountered While Trying To Open File. Please Contact Nutek For A Possible Solution.'),(sAlmText:='File Read Error While Reading Retain File',sRcyText:='An Error Was Encountered While Trying To Read File. Please Contact Nutek For A Possible Solution.'),(sAlmText:='File Close Error While Reading Retain File',sRcyText:='An Error Was Encountered While Trying To Close File. Please Contact Nutek For A Possible Solution.'),(sAlmText:='File Open Error While Writting Retain File',sRcyText:='An Error Was Encountered While Trying To Open File. Please Contact Nutek For A Possible Solution.'),(sAlmText:='File Create Error While Writting Retain File',sRcyText:='An Error Was Encountered While Trying To Create File. Please Contact Nutek For A Possible Solution.'),(sAlmText:='File Write Error While Writting Retain File',sRcyText:='An Error Was Encountered While Trying To Write File. Please Contact Nutek For A Possible Solution.'),(sAlmText:='File Close Error While Writting Retain File',sRcyText:='An Error Was Encountered While Trying To Close File. Please Contact Nutek For A Possible Solution.'),(sAlmText:='Directory Does Not Exist While Writing Retain File',sRcyText:='The Directory Does Not Exist. Please Contact Nutek For A Possible Solution.'),(sAlmText:='Revoke Board Available Request To Send From Supervisory Hermes',sRcyText:='Sending Illegal Message.'),(sAlmText:='Stop Transport Request To Send From Supervisory Hermes',sRcyText:='Sending Illegal Message.'),(sAlmText:='Transport Finished Request To Send From Supervisory Hermes',sRcyText:='Sending Illegal Message.'),(sAlmText:='Board Available Request To Send From Supervisory Hermes',sRcyText:='Sending Illegal Message.'),6(0),(sAlmText:='Check Alive Time Out',sRcyText:='Timeout Expired Before Operation Completed. Reset And Resume Operation.'),(sAlmText:='Waiting Check Alive Time Out',sRcyText:='Timeout Expired Before Operation Completed. Reset And Resume Operation.'),(sAlmText:='Check Alive Id Mismatch',sRcyText:='The Check Alive Id Value Does Not Match. Change The Value And Resend The Value.'),(sAlmText:='Machine Ready Request To Send From Supervisory Hermes',sRcyText:='Sending Illegal Message.'),(sAlmText:='Revoke Machine Ready Request To Send From Supervisory Hermes',sRcyText:='Sending Illegal Message.'),(sAlmText:='Start Transport Request To Send From Supervisory Hermes',sRcyText:='Sending Illegal Message.'),(sAlmText:='Set Configuration Request To Send From Supervisory Hermes',sRcyText:='Sending Illegal Message.'),(sAlmText:='Get Configuration Request To Send From Supervisory Hermes',sRcyText:='Sending Illegal Message.'),(sAlmText:='Current Configuration Request To Send From Supervisory Hermes',sRcyText:='Sending Illegal Message.'),(sAlmText:='Board Forecast Request To Send From Supervisory Hermes',sRcyText:='Sending Illegal Message.'),(sAlmText:='Query Board Info Request To Send From Supervisory Hermes',sRcyText:='Sending Illegal Message.'),(sAlmText:='Invalid Ident While Sending Data',sRcyText:='Invalid Ident Value.'),(sAlmText:='TCP Retry Send Data Error While Sending Data',sRcyText:='Problem Occurred In The TCP/IP Connection. Check The Connection And Try To Reconnect.'),(sAlmText:='TCP Send Data Error',sRcyText:='Problem Occurred In The TCP/IP Connection. Check The Connection And Try To Reconnect.'),(sAlmText:='Invalid Ident While Closing TCP',sRcyText:='Invalid Ident Value.'),(sAlmText:='Closing TCP Error',sRcyText:='Problem Occurred In The TCP/IP Connection. Check The Connection And Try To Reconnect.'),(sAlmText:='File Open Error While Writing Log',sRcyText:='An Error Was Encountered While Trying To Open File. Please Contact Nutek For A Possible Solution.'),(sAlmText:='File Create Error While Writing Log',sRcyText:='An Error Was Encountered While Trying To Create File. Please Contact Nutek For A Possible Solution.'),(sAlmText:='Get File Info Error While Writing Log',sRcyText:='An Error Was Encountered While Getting File Info. Please Contact Nutek For A Possible Solution.'),(sAlmText:='File Write Error While Writing Log',sRcyText:='An Error Was Encountered While Trying To Write File. Please Contact Nutek For A Possible Solution.'),(sAlmText:='File Close Error While Writing Log',sRcyText:='An Error Was Encountered While Trying To Close File. Please Contact Nutek For A Possible Solution.'),(sAlmText:='Directory Does Not Exist While Writing Log',sRcyText:='The Directory Does Not Exist.Please Contact Nutek For A Possible Solution.'),(sAlmText:='Invalid Ident While Closing TCP',sRcyText:='Invalid Ident Value.'),(sAlmText:='Closing TCP Error',sRcyText:='Problem Occurred In The TCP/IP Connection. Check The Connection And Try To Reconnect.'),3(0),(sAlmText:='Send Board Info Request To Send From Supervisory Hermes',sRcyText:='Sending Illegal Message.'),(sAlmText:='Query Work Order Info Request To Send From Supervisory Hermes',sRcyText:='Sending Illegal Message.'),(sAlmText:='Send Work Order Info Request To Send From Supervisory Hermes',sRcyText:='Sending Illegal Message.'),(sAlmText:='Board Arrived Request To Send From Supervisory Hermes',sRcyText:='Sending Illegal Message.'),(sAlmText:='Board Depated Request To Send From Supervisory Hermes',sRcyText:='Sending Illegal Message.'),(sAlmText:='QueryId Mismatch While Checking SendWorkOrderInfo and QueryWorkOrderInfo',sRcyText:='The QueryId Value Does Not Match. Change The Value And Resend The Value.'),(sAlmText:='QueryId Missing While Checking Send Work Order Info',sRcyText:='Missing Input Value For QueryId. Fill Up The Value And Resend.'),20(0),(sAlmText:='File Open Error While Writing Config File',sRcyText:='An Error Was Encountered While Trying To Open File. Please Contact Nutek For A Possible Solution.'),(sAlmText:='File Create Error While Writing Config File',sRcyText:='An Error Was Encountered While Trying To Create File. Please Contact Nutek For A Possible Solution.'),(sAlmText:='File Write Error While Writing Config File',sRcyText:='An Error Was Encountered While Trying To Write File. Please Contact Nutek For A Possible Solution.'),(sAlmText:='File Close Error While Writing Config File',sRcyText:='An Error Was Encountered While Trying To Close File. Please Contact Nutek For A Possible Solution.'),(sAlmText:='Directory Does Not Exist While Writing Config File',sRcyText:='The Directory Does Not Exist. Please Contact Nutek For A Possible Solution.'),9(0)];
END_VAR
(**)
(*Local Output*)
VAR
	bConnected : BOOL;
	bTest : BOOL;
	bTest1 : BOOL;
	bTest2 : BOOL;
	bHandshakeDone : BOOL;
	sInternalSnd : STRING[65535];
	bFileNotFound : BOOL := FALSE;
	bWriteConfig : BOOL := FALSE;
	bUpdateUIData : BOOL := FALSE;
END_VAR
(**)
(*Local Input*)
VAR
	udiRstErr : UDINT := 0;
	bPrep : BOOL := TRUE;
	bEn : BOOL := TRUE;
	bDis : BOOL := FALSE;
	tyParam : tyHermesSvyParam;
	sIPAddr : STRING[15] := '192.168.0.100';
	a_usiMacAddr : ARRAY[0..5] OF USINT := [6(0)];
	tyDTStructure : DTStructure := (year:=2020,month:=11,day:=05,wday:=05,hour:=21,minute:=28,second:=30,millisec:=123,microsec:=456);
	dtCurrDT : DATE_AND_TIME := DT#2019-02-23-12:30:50;
	sMcId : STRING[80] := '';
	sMagazineId : STRING[80] := '';
	iSlotId : INT;
	sBarcode : STRING[254] := '';
	eBoardTransfer1 : eHermesBoardTransfer := HermesTransferred;
	eBoardTransfer2 : eHermesBoardTransfer := HermesTransferred;
	eBoardTransfer3 : eHermesBoardTransfer := HermesTransferred;
	eBoardTransfer4 : eHermesBoardTransfer := HermesTransferred;
	sVersion : STRING[7] := '1.3';
	sWorkOrderId : STRING[80] := '';
	sBatchId : STRING[80] := '';
	sRecipeNm : STRING[254] := '';
	udiSndBffrSize : UDINT := 65536;
	udiRcvBffrSize : UDINT := 65536;
	udiAliveIdleTimeInSec : UDINT := 5;
	tConnTimeOut : TIME := T#30s;
	diTransferInTO : DINT := 30000;
	bNewBrdAvl : BOOL := FALSE;
	bOpsRun : BOOL := FALSE;
	udiFileKeepDay : UDINT := 30;
	sConfigFileName : STRING[80] := 'SvyHermes.dat';
	sProgNm : STRING[15] := 'SvyHermes';
	sRetainFileName : STRING[80] := 'WorkOrder.dat';
	bNtSettingsLoadDone : BOOL := TRUE;
	bSvyPrep : BOOL := FALSE;
	bSvyEn : BOOL := FALSE;
	sInfoMsg : STRING[200];
	sInfoMsg1 : STRING[200];
	sInfoMsg2 : STRING[200];
	sInfoMsg3 : STRING[200];
	sInfoMsg4 : STRING[200];
	sInfoMsg5 : STRING[200];
	sInfoMsg6 : STRING[200];
	bEndSen : BOOL := FALSE;
	tyHermesCurrConfiguration : tyHermesConfiguration;
	bQueryWorkOrderInfo : BOOL;
	bReinsertBrd : BOOL;
	bManualInsertData : BOOL;
	bQueryInsertBoard : BOOL;
	bAcceptCondition : BOOL;
	bAllZonesEmpty : BOOL;
	bDeleteWorkOrder : BOOL;
	bFirstMcIntheLine : BOOL;
	bUSHermesStopTransportSnd1 : BOOL;
	bUSHermesStopTransportSnd2 : BOOL;
	bUSHermesStopTransportSnd3 : BOOL;
	bUSHermesStopTransportSnd4 : BOOL;
	bDSHermesTransportFinishedSnd1 : BOOL;
	bDSHermesTransportFinishedSnd2 : BOOL;
	bDSHermesTransportFinishedSnd3 : BOOL;
	bDSHermesTransportFinishedSnd4 : BOOL;
	tyUSHermesBoardArrivedData1 : tyHermesBoardAvailable;
	tyUSHermesBoardArrivedData2 : tyHermesBoardAvailable;
	tyUSHermesBoardArrivedData3 : tyHermesBoardAvailable;
	tyUSHermesBoardArrivedData4 : tyHermesBoardAvailable;
	tyDSHermesBoardDepartedData1 : tyHermesBoardAvailable;
	tyDSHermesBoardDepartedData2 : tyHermesBoardAvailable;
	tyDSHermesBoardDepartedData3 : tyHermesBoardAvailable;
	tyDSHermesBoardDepartedData4 : tyHermesBoardAvailable;
	bInternalUse : BOOL;
	sInternalRcv : STRING[65535];
END_VAR
(**)
(*Local*)
VAR
	bRstErr : BOOL;
	udiRstErrOld : UDINT;
	bInitDone : BOOL;
	bInitialDone : BOOL;
	bRun : BOOL;
	bStop : BOOL;
	bRstConnection : BOOL;
	bRstState : BOOL;
	bRcvWorkOrderInfo1 : BOOL;
	bRcvWorkOrderInfo2 : BOOL;
	bRcvInsertBoardInfo : BOOL;
	bRstWorkOrderInfo : BOOL;
	bReplyWorkOrderInfo : BOOL := FALSE;
	bFoundIndexUS1 : BOOL;
	bFoundIndexUS2 : BOOL;
	bFoundIndexUS3 : BOOL;
	bFoundIndexUS4 : BOOL;
	bFoundIndexDS1 : BOOL;
	bFoundIndexDS2 : BOOL;
	bFoundIndexDS3 : BOOL;
	bFoundIndexDS4 : BOOL;
	udiFoundIndexUS1 : UDINT;
	udiFoundIndexUS2 : UDINT;
	udiFoundIndexUS3 : UDINT;
	udiFoundIndexUS4 : UDINT;
	udiFoundIndexDS1 : UDINT;
	udiFoundIndexDS2 : UDINT;
	udiFoundIndexDS3 : UDINT;
	udiFoundIndexDS4 : UDINT;
	k : UDINT := 0;
	kk : UDINT := 0;
	j : INT := 1;
	jj : INT := 2;
	jjj : INT := 3;
	jjjj : INT := 4;
	udiSvrIdent : UDINT;
	udiClntIdent : UDINT;
	udiClntIdentExtra : UDINT;
	udiXMLTableWriteIdx : UDINT;
	udiMsgSendBffr : UDINT;
	udiSndMsgLen : UDINT;
	sSnd : STRING[65535];
	sRcv : STRING[65535];
	a_tyXMLTableDataRcv : ARRAY[0..200] OF tyXMLTableDat;
	a_tyXMLTableDataSnd : ARRAY[0..200] OF tyXMLTableDat;
	a_eMsgSend : ARRAY[0..50] OF eHermesMsgType;
	tyMsgTypeRcv : tyHermesMsgType;
	tyCheckAliveSnd : tyHermesCheckAlive;
	tyCheckAlivePingSnd : tyHermesCheckAlive;
	tyCheckAlivePongSnd : tyHermesCheckAlive;
	tyCheckAliveRcv : tyHermesCheckAlive;
	tyCheckAlivePingRcv : tyHermesCheckAlive;
	tyCheckAlivePongRcv : tyHermesCheckAlive;
	tyServiceDescriptionRcv : tyHermesServiceDescription;
	tySServiceDescriptionSnd : tyHermesSServiceDescription;
	tySServiceDescriptionRcv : tyHermesSServiceDescription;
	tyNotificationSnd : tyHermesNotification;
	tyNotificationRcv : tyHermesNotification;
	tyBoardAvailableRcv : tyHermesBoardAvailable;
	tyMachineReady : tyHermesMachineReady;
	tyStartTransport : tyHermesStartTransport;
	tyStopTransport : tyHermesStopTransport;
	tyTransportFinished : tyHermesTransportFinished;
	tySetConfiguration : tyHermesSetConfiguration;
	tySetConfigurationRcv : tyHermesSetConfiguration;
	tySetConfigurationModified : tyHermesSetConfiguration;
	tyCurrentConfigurationRcv : tyHermesCurrentConfiguration;
	tyCurrentConfigurationSnd : tyHermesCurrentConfiguration;
	tyBoardForecast : tyHermesBoardForecast;
	tyBoardArrivedRcv : tyHermesBoardArrived;
	tyBoardArrived1 : tyHermesBoardArrived;
	tyBoardArrived2 : tyHermesBoardArrived;
	tyBoardArrived3 : tyHermesBoardArrived;
	tyBoardArrived4 : tyHermesBoardArrived;
	tyBoardDepartedRcv : tyHermesBoardDeparted;
	tyBoardDeparted1 : tyHermesBoardDeparted;
	tyBoardDeparted2 : tyHermesBoardDeparted;
	tyBoardDeparted3 : tyHermesBoardDeparted;
	tyBoardDeparted4 : tyHermesBoardDeparted;
	tyQueryBoardInfo : tyHermesQueryBoardInfo;
	tySendBoardInfo : tyHermesSendBoardInfo;
	tyQueryWorkOrderInfo : tyHermesQueryWorkOrderInfo;
	tySendWorkOrderInfoAcc : tyHermesSendWorkOrderInfo;
	tySendWorkOrderInfoRcv : tyHermesSendWorkOrderInfo;
	tyReplyWorkOrderInfo : tyHermesReplyWorkOrderInfo;
	fbCreateSvr : fbTCPCreateSvr;
	fbListen : fbTCPListen;
	fbRcv : fbTCPRcv;
	fbSend : fbTCPSnd;
	fbCloseSvr : fbTCPClose;
	fbCloseClnt : fbTCPClose;
	fbParseXMLTable : fbHermesParseXMLTable;
	fbCheckAlive : fbHermesCheckAlive;
	fbCheckAliveSendPing : fbHermesCheckAliveSendPing;
	fbCheckAliveRcvPing : fbHermesCheckAliveRcvPing;
	fbSequenceSvy : fbHermesSequenceSvy;
	fbSequenceTO : fbHermesSequenceSvyTO;
	eStatOld : eHermesAction := HermesActIdle;
	tyParamOld : tyHermesSvyParam;
	udiLogCntr : UDINT := 1;
	udiWriteLogCntr : UDINT := 1;
	a_sLogList : ARRAY[1..10] OF STRING[65535];
	sDT : STRING[80];
	dtCurrDTTemp : DATE_AND_TIME;
	fbFileAppend1 : fbFileFullAppend;
	fbFileOldDel1 : fbFileOldDel;
	fbFileRead1 : fbFileFullRead;
	fbFileWrite1 : fbFileFullWrite;
	fbDelayTm : TON;
	fbDelayTm1 : TON;
	udiTargetAddress : UDINT := 0;
	udiTargetAddress1 : UDINT := 0;
	udiSizeAddress : UDINT := 0;
	udiSizeAddress1 : UDINT := 0;
	udiRetainDataAddr : UDINT;
	udiRetainDataLen : UDINT;
	diReqWidthInUM : DINT;
	iWriteLogStep : INT := 0;
	udiModuleNum : UDINT := 6651;
END_VAR
```

#### Act_Background_QueryWorkOrderInfo1.st - not listed in the package file held
```iecst
(** 2021-08-01 **)
ACTION Act_Background_QueryWorkOrderInfo1:

	IF EDGEPOS(p_bQueryWorkOrderInfo) THEN

		fHermesAddOneMsgSend(ADR(a_eMsgSend) , ADR(udiMsgSendBffr) , HermesMsgTypeQueryWorkOrderInfo);

		fHermesGenerateUUID(ADR(tyQueryWorkOrderInfo.tyData.sQueryId) , p_tyDTStructure , pa_usiMacAddr); //Generate QueryID

		tyQueryWorkOrderInfo.tyData.sMachineId							:= p_sMcId;
		tyQueryWorkOrderInfo.tyData.sMagazineId							:= p_sMagazineId;
		tyQueryWorkOrderInfo.tyData.iSlotId								:= p_iSlotId;
		tyQueryWorkOrderInfo.tyData.sBarcode						    := p_sBarcode;

		tyQueryWorkOrderInfo.tyAvl.bQueryId							    := tyQueryWorkOrderInfo.tyData.sQueryId <> '';
		tyQueryWorkOrderInfo.tyAvl.bMachineId							:= tyQueryWorkOrderInfo.tyData.sMachineId <> '';
		tyQueryWorkOrderInfo.tyAvl.bMagazineId							:= tyQueryWorkOrderInfo.tyData.sMagazineId <> '';
		tyQueryWorkOrderInfo.tyAvl.bSlotId								:= tyQueryWorkOrderInfo.tyData.iSlotId <> 0;
		tyQueryWorkOrderInfo.tyAvl.bBarcode								:= tyQueryWorkOrderInfo.tyData.sBarcode <> '';

		tyQueryQueue[usiQueueIdx].usiPriority := 0;
		tyQueryQueue[usiQueueIdx].udiTracedSubjectAddr := ADR(bhvBrd);
		tyQueryQueue[usiQueueIdx].tyQueryWorkOrder := tyQueryWorkOrderInfo;
		usiQueueIdx := usiQueueIdx +1;
	END_IF

	FOR usidx:= 0 TO usiQueueIdxDO DO

	END_FOR

END_ACTION
```

### LF.typ - Do Not Change!!!
```iecst
(*2019-04-25*)
(**)
(*Action*)

TYPE
	eLFAction :
		(
		LFActIdle,
		LFActBGStartRun,
		LFActBGStopRun,
		LFActSyncPLCTm,
		LFActChgAllAuto,
		LFActChgAllMnl,
		LFActChgSeqAuto,
		LFActChgSeqMnl
		);
	eLFOPCUAStep :
		(
		LFOPCUAStepIncCntr,
		LFOPCUAStepChkHdls,
		LFOPCUAStepConnect,
		LFOPCUAStepWriteHdls,
		LFOPCUAStepReadHdls,
		LFOPCUAStepWrite,
		LFOPCUAStepRead,
		LFOPCUAStepStopChk
		);
	tyOPCUAHdlList : 	STRUCT
		a_dwHdls : ARRAY[0..MAX_INDEX_NODELIST]OF DWORD;
	END_STRUCT;
END_TYPE
```

### LFLeader.var - Change By Project
```iecst
(*2019-04-30*)
(**)
(*Action & State & Status*)
VAR
	p_LFLeaderStat : UDINT;
	p_LFLeaderStatus : UDINT;
	p_LFLeaderStatTxt : UDINT;
END_VAR
(**)
(*Alarm*)
VAR
	p_LFLeaderAlmData : UDINT;
END_VAR
(**)
(*Output*)
VAR
	p_LFLeaderFollowerInfo : UDINT;
	p_LFLeaderFollowerToLeaderTag : UDINT;
END_VAR
```

### Program Logical/LF/LFLeader (IEC, version 1.00.0) - 1.00.0 - NtHermes v5.00.0 , NtTCP v5.00.0 , NtMessage v5.00.0

#### Init.st - Change By Project
```iecst
(** 2019-04-30 **)
PROGRAM _INIT

	(* Always Change If Project Change *)

	//Pass Address To Global Address For External Use
	//Action, State & Status
	p_LFLeaderStat		:= ADR(eStat);
	p_LFLeaderStatus	:= ADR(eStatus);
	p_LFLeaderStatTxt	:= ADR(sStatTxt);

	//Alarm
	p_LFLeaderAlmData	:= ADR(tyAlmData);

	//Output
	p_LFLeaderFollowerInfo			:= ADR(a_tyFollowerInfo);
	p_LFLeaderFollowerToLeaderTag	:= ADR(a_tyFollowerToLeaderTag);

	(* Always Change If Project Change *)

END_PROGRAM
```

#### Act_InitGlobal.st - Change By Project
```iecst
(** 2020-08-06 **)
ACTION Act_InitGlobal:

	(* Always Change If Project Change *)

	//Pass Data To Link
	p_bLinkStartupRun ACCESS p_StartupRun;
	p_bLinkNtParamLFPrep ACCESS p_NtParamLFPrep;
	p_bLinkNtParamLeaderMc ACCESS p_NtParamLeaderMc;
	p_bLinkNtParamLFUsrSetPrep ACCESS p_NtParamLFUsrSetPrep;
	p_bLinkMcParamLFLeaderMc ACCESS p_McParamLFLeaderMc;
	p_bLinkUILeaderRun ACCESS p_UILeaderRun;

	//Pass Data To Internal Use
	p_eAct ACCESS p_UILFLeaderAct;
	p_udiRstErr ACCESS p_RstErrReset;
	p_bEn ACCESS p_McParamLFEn;
	p_sReqProdRcpNm ACCESS p_ProdRcpCurrRcp0Nm;
//	p_diReqProdWidth ACCESS p_ProdRcpCurrRcp0Width;
	p_diBeforeOven ACCESS p_McParamLFMcIdxBeforeOven;
	p_diAfterOven ACCESS p_McParamLFMcIdxAfterOven;
	p_tOnlineChkDlyTm ACCESS p_NtParamLFLeaderOnlineChkDlyTm;
	p_tSetTmOffDlyTm ACCESS p_NtParamLFLeaderSetTmOffDlyTm;
	p_dtCurrDT ACCESS p_TimeCurrDT;
	pa_sLFIPAddr ACCESS p_McParamLFIPAddr;
	pa_bLFOnline ACCESS p_McParamLFOnline;
	p_sProgNm ACCESS p_NtParamLFLeaderProgNm;
	p_bNtSettingsLoadDone ACCESS p_StartupNtSettingsLoadDone;

	p_diBeforeOven2 ACCESS p_McParamLFMcIdxBeforeOven2;		// ADD
	p_diAfterOven2 ACCESS p_McParamLFMcIdxAfterOven2;		//

	p_bWidth2Prep ACCESS p_NtParamLFWidth2Prep;
	p_bLFSeqStayActive ACCESS p_McParamLFSeqStayActive;

	(* Always Change If Project Change *)

END_ACTION
```

#### InputRef_Link.var - Change By Project
```iecst
(*2019-04-25*)
(**)
VAR
	p_bLinkStartupRun : REFERENCE TO BOOL;
	p_bLinkNtParamLFPrep : REFERENCE TO BOOL;
	p_bLinkNtParamLeaderMc : REFERENCE TO BOOL;
	p_bLinkNtParamLFUsrSetPrep : REFERENCE TO BOOL;
	p_bLinkMcParamLFLeaderMc : REFERENCE TO BOOL;
	p_bLinkUILeaderRun : REFERENCE TO BOOL;
	bUILeaderStart : BOOL;
	bUILeaderStop : BOOL;
END_VAR
```

#### Act_LinkAction.st - Change By Project
```iecst
(** 2019-04-25 **)
ACTION Act_LinkAction:

	IF (p_bLinkUILeaderRun = TRUE) AND ((bRun1 = FALSE) OR (bRun2 = FALSE)) THEN
		bUILeaderStart	:= TRUE;
		bUILeaderStop	:= FALSE;
	END_IF

	IF (p_bLinkUILeaderRun = FALSE) AND ((bRun1 = TRUE) OR (bRun2 = TRUE)) THEN
		bUILeaderStart	:= FALSE;
		bUILeaderStop	:= TRUE;
	END_IF

	IF bUILeaderStart = TRUE THEN
		p_eAct	:= LFActBGStartRun;

		IF (eStat = LFActBGStartRun) AND (eStatus = Done) THEN
			p_eAct			:= LFActIdle;
			bUILeaderStart	:= FALSE;
		END_IF

	ELSIF bUILeaderStop = TRUE THEN
		p_eAct	:= LFActBGStopRun;

		IF (eStat = LFActBGStopRun) AND (eStatus = Done) THEN
			p_eAct			:= LFActIdle;
			bUILeaderStop	:= FALSE;
		END_IF

	END_IF

END_ACTION
```

#### Act_LinkEn.st - Change By Project
```iecst
(** 2019-04-25 **)
ACTION Act_LinkEn:

	//Link bPrep, bEn & bDis
	p_bPrep	:= p_bLinkNtParamLFPrep;
	p_bDis	:= p_bLinkStartupRun OR (NOT p_bLinkNtParamLFUsrSetPrep AND NOT p_bLinkNtParamLeaderMc) OR (p_bLinkNtParamLFUsrSetPrep AND NOT p_bLinkMcParamLFLeaderMc);

END_ACTION
```

#### Act_Link.st - Change By Project
```iecst
(** 2020-08-06 **)
ACTION Act_Link:
	IF p_bWidth2Prep THEN
		p_diReqProdWidth ACCESS p_ProdRcpCurrRcp0Width2;
	ELSE
		p_diReqProdWidth ACCESS p_ProdRcpCurrRcp0Width;
	END_IF

END_ACTION
```

#### Cyclic.st - Do Not Change!!!
```iecst
(** 2019-04-23 **)
PROGRAM _CYCLIC

	IF bInitDone = FALSE THEN
		bInitDone	:= TRUE;

		Act_InitLocal;
		Act_InitGlobal;

	ELSIF bInitialDone = FALSE THEN
		IF p_bNtSettingsLoadDone = TRUE THEN
			bInitialDone	:= TRUE;

			Act_Initial;
		END_IF

	ELSE

		Act_RstErr;
		Act_LinkAction;
		Act_Action;
		Act_LinkEn;

		IF (p_bPrep = TRUE) AND (p_bEn = TRUE) AND (p_bDis = FALSE) THEN
			Act_Link;
			Act_Background;
			Act_Main;

		ELSE
			Act_Main_Disable;

			IF eStat <> LFActIdle THEN
				eStatus	:= Done;
			ELSE
				eStatus	:= Idle;
			END_IF
		END_IF

		Act_Alarm;

	END_IF

END_PROGRAM
```

#### Act_RstErr.st - Do Not Change!!!
```iecst
(** 2019-04-23 **)
ACTION Act_RstErr:

	IF p_udiRstErr <> udiRstErrOld THEN
		bRstErr			:= TRUE;
		udiRstErrOld	:= p_udiRstErr;
	ELSE
		bRstErr			:= FALSE;
	END_IF

END_ACTION
```

#### Act_InitLocal.st - Do Not Change!!!
```iecst
(** 2020-08-06 **)
ACTION Act_InitLocal:

	//Input Reference Link To Local Variable
	p_eAct ACCESS ADR(eAct);
	p_udiRstErr ACCESS ADR(udiRstErr);
	p_bPrep ACCESS ADR(bPrep);
	p_bEn ACCESS ADR(bEn);
	p_bDis ACCESS ADR(bDis);
	p_sReqProdRcpNm ACCESS ADR(sReqProdRcpNm);
	p_diReqProdWidth ACCESS ADR(diReqProdWidth);
	p_sReqMagRcpNm ACCESS ADR(sReqMagRcpNm);
	p_diBeforeOven ACCESS ADR(diBeforeOven);
	p_diAfterOven ACCESS ADR(diAfterOven);
	p_diBeforeOven2 ACCESS ADR(diBeforeOven2);
	p_diAfterOven2 ACCESS ADR(diAfterOven2);
	p_tOnlineChkDlyTm ACCESS ADR(tOnlineChkDlyTm);
	p_tSetTmOffDlyTm ACCESS ADR(tSetTmOffDlyTm);
	p_dtCurrDT ACCESS ADR(dtCurrDT);
	pa_sLFIPAddr ACCESS ADR(a_sLFIPAddr);
	pa_bLFOnline ACCESS ADR(a_bLFOnline);
	p_sLeaderProgTagNm ACCESS ADR(sLeaderProgTagNm);
	p_sFollowerProgTagNm ACCESS ADR(sFollowerProgTagNm);
	p_sProgNm ACCESS ADR(sProgNm);
	p_bNtSettingsLoadDone ACCESS ADR(bNtSettingsLoadDone);
	p_bWidth2Prep ACCESS ADR(bWidth2Prep);
//	p_bLFSeqStayActive ACCESS ADR(bLFSeqStayActive);

END_ACTION
```

#### Act_Initial.st - Do Not Change!!!
```iecst
(** 2020-10-05 **)
ACTION Act_Initial:

	//Initial
	sStatTxt	:= a_sStatText[eStat];

	fbOnlineChk.pa_tyLeaderToFollowerTag	:= ADR(a_tyLeaderToFollowerTag);
	fbOnlineChk.pa_tyFollowerInfo	:= ADR(a_tyFollowerInfo);
	fbOnlineChk.tDlyTm				:= p_tOnlineChkDlyTm;
	fbOnlineChk(bEn := FALSE);

	fbSyncTm.pa_tyLeaderToFollowerTag	:= ADR(a_tyLeaderToFollowerTag);
	fbSyncTm.tDlyTm						:= p_tSetTmOffDlyTm;
	fbSyncTm(bEn := FALSE);

	fbChgAll.pa_tyLeaderToFollowerTag	:= ADR(a_tyLeaderToFollowerTag);
	fbChgAll(bEn := FALSE);

	fbChgSeq.pa_tyLeaderToFollowerTag	:= ADR(a_tyLeaderToFollowerTag);
	fbChgSeq(bEn := FALSE);

	fbBlkUSDS.pa_tyLeaderToFollowerTag	:= ADR(a_tyLeaderToFollowerTag);
	fbBlkUSDS(bEn := FALSE);

	fbDataUpdt.pa_tyLeaderToFollowerTag	:= ADR(a_tyLeaderToFollowerTag);
	fbDataUpdt(bEn := FALSE);

	fbConnect.tyOPCUAParam.sPort	:= '4840';
	fbConnect(bEn := FALSE);

	fbGetNodeHdlListWr.uiTagNmCnt			:= 17;
	fbGetNodeHdlListWr.a_sServerTagNm[0]	:= CONCAT(CONCAT('::' , p_sFollowerProgTagNm) , ':tyLeaderToFollowerTag.sReqProdRcpNm');
	fbGetNodeHdlListWr.a_sServerTagNm[1]	:= CONCAT(CONCAT('::' , p_sFollowerProgTagNm) , ':tyLeaderToFollowerTag.diReqProdRcpWidth');
	fbGetNodeHdlListWr.a_sServerTagNm[2]	:= CONCAT(CONCAT('::' , p_sFollowerProgTagNm) , ':tyLeaderToFollowerTag.sReqMagRcpNm');
	fbGetNodeHdlListWr.a_sServerTagNm[3]	:= CONCAT(CONCAT('::' , p_sFollowerProgTagNm) , ':tyLeaderToFollowerTag.bMnlAccData');
	fbGetNodeHdlListWr.a_sServerTagNm[4]	:= CONCAT(CONCAT('::' , p_sFollowerProgTagNm) , ':tyLeaderToFollowerTag.bBypassMnlAccData');
	fbGetNodeHdlListWr.a_sServerTagNm[5]	:= CONCAT(CONCAT('::' , p_sFollowerProgTagNm) , ':tyLeaderToFollowerTag.bBlkDS');
	fbGetNodeHdlListWr.a_sServerTagNm[6]	:= CONCAT(CONCAT('::' , p_sFollowerProgTagNm) , ':tyLeaderToFollowerTag.bBlkUS');
	fbGetNodeHdlListWr.a_sServerTagNm[7]	:= CONCAT(CONCAT('::' , p_sFollowerProgTagNm) , ':tyLeaderToFollowerTag.bSetTm');
	fbGetNodeHdlListWr.a_sServerTagNm[8]	:= CONCAT(CONCAT('::' , p_sFollowerProgTagNm) , ':tyLeaderToFollowerTag.dtTm');
	fbGetNodeHdlListWr.a_sServerTagNm[9]	:= CONCAT(CONCAT('::' , p_sFollowerProgTagNm) , ':tyLeaderToFollowerTag.uiTmZone');
	fbGetNodeHdlListWr.a_sServerTagNm[10]	:= CONCAT(CONCAT('::' , p_sFollowerProgTagNm) , ':tyLeaderToFollowerTag.bBypassWidthChk');
	fbGetNodeHdlListWr.a_sServerTagNm[11]	:= CONCAT(CONCAT('::' , p_sFollowerProgTagNm) , ':tyLeaderToFollowerTag.usiRunTm');
	fbGetNodeHdlListWr.a_sServerTagNm[12]	:= CONCAT(CONCAT('::' , p_sFollowerProgTagNm) , ':tyLeaderToFollowerTag.bProdNameUSWarn');
	fbGetNodeHdlListWr.a_sServerTagNm[13]	:= CONCAT(CONCAT('::' , p_sFollowerProgTagNm) , ':tyLeaderToFollowerTag.bProdNameDSWarn');
	fbGetNodeHdlListWr.a_sServerTagNm[14]	:= CONCAT(CONCAT('::' , p_sFollowerProgTagNm) , ':tyLeaderToFollowerTag.bProdWidthUSWarn');
	fbGetNodeHdlListWr.a_sServerTagNm[15]	:= CONCAT(CONCAT('::' , p_sFollowerProgTagNm) , ':tyLeaderToFollowerTag.bProdWidthDSWarn');
	fbGetNodeHdlListWr.a_sServerTagNm[16]	:= CONCAT(CONCAT('::' , p_sFollowerProgTagNm) , ':tyLeaderToFollowerTag.bLeaderSeqCtrlInActive');
	fbGetNodeHdlListWr(bEn := FALSE);

	fbGetNodeHdlListRd.uiTagNmCnt			:= 14;
	fbGetNodeHdlListRd.a_sServerTagNm[0]	:= CONCAT(CONCAT('::' , p_sFollowerProgTagNm) , ':tyFollowerToLeaderTag.sCurrProdRcp');
	fbGetNodeHdlListRd.a_sServerTagNm[1]	:= CONCAT(CONCAT('::' , p_sFollowerProgTagNm) , ':tyFollowerToLeaderTag.diCurrProdWidthUS');
	fbGetNodeHdlListRd.a_sServerTagNm[2]	:= CONCAT(CONCAT('::' , p_sFollowerProgTagNm) , ':tyFollowerToLeaderTag.sCurrMagRcp');
	fbGetNodeHdlListRd.a_sServerTagNm[3]	:= CONCAT(CONCAT('::' , p_sFollowerProgTagNm) , ':tyFollowerToLeaderTag.sIPAddr');
	fbGetNodeHdlListRd.a_sServerTagNm[4]	:= CONCAT(CONCAT('::' , p_sFollowerProgTagNm) , ':tyFollowerToLeaderTag.sMcNm');
	fbGetNodeHdlListRd.a_sServerTagNm[5]	:= CONCAT(CONCAT('::' , p_sFollowerProgTagNm) , ':tyFollowerToLeaderTag.bSectionLeader');
	fbGetNodeHdlListRd.a_sServerTagNm[6]	:= CONCAT(CONCAT('::' , p_sFollowerProgTagNm) , ':tyFollowerToLeaderTag.usiRunTm');
	fbGetNodeHdlListRd.a_sServerTagNm[7]	:= CONCAT(CONCAT('::' , p_sFollowerProgTagNm) , ':tyFollowerToLeaderTag.bProdRcpErr');
	fbGetNodeHdlListRd.a_sServerTagNm[8]	:= CONCAT(CONCAT('::' , p_sFollowerProgTagNm) , ':tyFollowerToLeaderTag.bProdWidthErr');
	fbGetNodeHdlListRd.a_sServerTagNm[9]	:= CONCAT(CONCAT('::' , p_sFollowerProgTagNm) , ':tyFollowerToLeaderTag.bMagRcpErr');
	fbGetNodeHdlListRd.a_sServerTagNm[10]	:= CONCAT(CONCAT('::' , p_sFollowerProgTagNm) , ':tyFollowerToLeaderTag.bSyncTmErr');
	fbGetNodeHdlListRd.a_sServerTagNm[11]	:= CONCAT(CONCAT('::' , p_sFollowerProgTagNm) , ':tyFollowerToLeaderTag.diCurrProdWidthDS');
	fbGetNodeHdlListRd.a_sServerTagNm[12]	:= CONCAT(CONCAT('::' , p_sFollowerProgTagNm) , ':tyFollowerToLeaderTag.eCurrMachineStat');
	fbGetNodeHdlListRd.a_sServerTagNm[13]	:= CONCAT(CONCAT('::' , p_sFollowerProgTagNm) , ':tyFollowerToLeaderTag.bProdChgOverActive');
	fbGetNodeHdlListRd(bEn := FALSE);

	fbWriteList.uiTagNmCnt	:= 17;
	fbWriteList(bEn := FALSE);

	fbReadList.uiTagNmCnt	:= 14;
	fbReadList(bEn := FALSE);

	fbDisconnect(bEn := FALSE);

END_ACTION
```

#### Act_Action.st - Do Not Change!!!
```iecst
(** 2019-04-23 **)
ACTION Act_Action:

	//Reset Error
	IF (eStatus = Error) AND bRstErr THEN
		p_eAct	:= LFActIdle;
		eStat	:= LFActIdle;
	END_IF

	//Set p_eAct
	IF eStatus = Idle OR eStatus = Busy OR eStatus = Done THEN
		eStat	:= p_eAct;
	END_IF

END_ACTION
```

#### Act_Main.st - Do Not Change!!!
```iecst
(** 2021-04-20 **)
ACTION Act_Main:

	IF eStatOld <> eStat THEN
		fbSyncTm(bEn := FALSE);
		fbChgAll(bEn := FALSE);
		fbChgSeq(bEn := FALSE);

		sStatTxt	:= a_sStatText[eStat];

		eStatOld	:= eStat;

		eStatus		:= Busy;
	END_IF

	//Main
	CASE eStat OF

		LFActIdle:
			eStatus	:= Idle;

		LFActBGStartRun:
			IF eStatus = Idle OR eStatus = Busy THEN

				bRun1		:= TRUE;
				bRun2		:= TRUE;
				bStop		:= FALSE;
				bStop1Done	:= FALSE;
				bStop2Done	:= FALSE;
				eStatus		:= Done;

			END_IF

		LFActBGStopRun:
			IF eStatus = Idle OR eStatus = Busy THEN

				eStatus	:= Busy;

				bStop	:= TRUE;

				IF bStop1Done AND bStop2Done THEN

					bRun1		:= FALSE;
					bRun2		:= FALSE;
					bStop		:= FALSE;
					bStop1Done	:= FALSE;
					bStop2Done	:= FALSE;
					eStatus		:= Done;

				END_IF

			END_IF

		LFActSyncPLCTm:
			IF eStatus = Idle OR eStatus = Busy THEN

				IF bRun1 AND bRun2 THEN
					eStatus	:= Busy;

					fbSyncTm.dtCurrDT		:= p_dtCurrDT;
					fbSyncTm.diMcNum		:= diMcNum;
					fbSyncTm(bEn := TRUE);

					IF fbSyncTm.udiStatus = 0 THEN
						eStatus	:= Done;
					ELSIF fbSyncTm.udiStatus < 65534 THEN
						eStatus		:= Error;
						udiStatus	:= fbSyncTm.udiStatus;
					END_IF

				ELSE
					eStatus		:= Error;
					udiStatus	:= 10000;	//Background Not Running While Calling Sync PLC Tm
				END_IF

			END_IF

		LFActChgAllAuto:
			IF eStatus = Idle OR eStatus = Busy THEN

				IF bRun1 AND bRun2 THEN
					eStatus	:= Busy;

					fbChgAll.bChgAuto					:= TRUE;
					fbChgAll.a_bOnline					:= pa_bLFOnline;;
					fbChgAll.a_tyFollowerToLeaderTag	:= a_tyFollowerToLeaderTag;
					fbChgAll.sReqProdRcpNm				:= p_sReqProdRcpNm;
					fbChgAll.diReqProdRcpWidth			:= p_diReqProdWidth;
					fbChgAll.sReqMagRcpNm				:= p_sReqMagRcpNm;
					fbChgAll.diMcNum					:= diMcNum;
					fbChgAll(bEn := TRUE);

					IF fbChgAll.udiStatus = 0 THEN
						eStatus	:= Done;
					ELSIF fbChgAll.udiStatus < 65534 THEN
						eStatus		:= Error;
						udiStatus	:= fbChgAll.udiStatus;
					END_IF

				ELSE
					eStatus		:= Error;
					udiStatus	:= 10001;	//Background Not Running While Changing All Recipe Automatically
				END_IF

			END_IF

		LFActChgAllMnl:
			IF eStatus = Idle OR eStatus = Busy THEN

				IF bRun1 AND bRun2 THEN
					eStatus	:= Busy;

					fbChgAll.bChgAuto					:= FALSE;
					fbChgAll.a_bOnline					:= pa_bLFOnline;
					fbChgAll.a_tyFollowerToLeaderTag	:= a_tyFollowerToLeaderTag;
					fbChgAll.sReqProdRcpNm				:= p_sReqProdRcpNm;
					fbChgAll.diReqProdRcpWidth			:= p_diReqProdWidth;
					fbChgAll.sReqMagRcpNm				:= p_sReqMagRcpNm;
					fbChgAll.diMcNum					:= diMcNum;
					fbChgAll(bEn := TRUE);

					IF fbChgAll.udiStatus = 0 THEN
						eStatus	:= Done;
					ELSIF fbChgAll.udiStatus < 65534 THEN
						eStatus		:= Error;
						udiStatus	:= fbChgAll.udiStatus;
					END_IF

				ELSE
					eStatus		:= Error;
					udiStatus	:= 10002;	//Background Not Running While Changing All Recipe Manually
				END_IF

			END_IF

		LFActChgSeqAuto:
			IF eStatus = Idle OR eStatus = Busy THEN

				IF bRun1 AND bRun2 THEN
					eStatus	:= Busy;

					fbChgSeq.bChgAuto					:= TRUE;
					fbChgSeq.a_bOnline					:= pa_bLFOnline;;
					fbChgSeq.a_tyFollowerToLeaderTag	:= a_tyFollowerToLeaderTag;
					fbChgSeq.sReqProdRcpNm				:= p_sReqProdRcpNm;
					fbChgSeq.diReqProdRcpWidth			:= p_diReqProdWidth;
					fbChgSeq.sReqMagRcpNm				:= p_sReqMagRcpNm;
					fbChgSeq.diMcNum					:= diMcNum;
					fbChgSeq(bEn := TRUE);

					IF fbChgSeq.udiStatus = 0 THEN
						eStatus	:= Done;
					ELSIF fbChgSeq.udiStatus < 65534 THEN
						eStatus		:= Error;
						udiStatus	:= fbChgSeq.udiStatus;
					END_IF

				ELSE
					eStatus		:= Error;
					udiStatus	:= 10003;	//Background Not Running While Changing Recipe In Sequence Automatically
				END_IF

			END_IF

		LFActChgSeqMnl:
			IF eStatus = Idle OR eStatus = Busy THEN

				IF bRun1 AND bRun2 THEN
					eStatus	:= Busy;

					fbChgSeq.bChgAuto					:= FALSE;
					fbChgSeq.a_bOnline					:= pa_bLFOnline;;
					fbChgSeq.a_tyFollowerToLeaderTag	:= a_tyFollowerToLeaderTag;
					fbChgSeq.sReqProdRcpNm				:= p_sReqProdRcpNm;
					fbChgSeq.diReqProdRcpWidth			:= p_diReqProdWidth;
					fbChgSeq.sReqMagRcpNm				:= p_sReqMagRcpNm;
					fbChgSeq.diMcNum					:= diMcNum;
					fbChgSeq(bEn := TRUE);

					IF fbChgSeq.udiStatus = 0 THEN
						eStatus	:= Done;
					ELSIF fbChgSeq.udiStatus < 65534 THEN
						eStatus		:= Error;
						udiStatus	:= fbChgSeq.udiStatus;
					END_IF

				ELSE
					eStatus		:= Error;
					udiStatus	:= 10004;	//Background Not Running While Changing Recipe In Sequence Manually
				END_IF

			END_IF

	END_CASE

END_ACTION
```

#### Act_Background.st - Do Not Change!!!
```iecst
(** 2019-04-25 **)
ACTION Act_Background:

	IF EDGEPOS(bRun1 AND bRun2) THEN

		FOR di := 1 TO c_diLFClntNum DO
			IF pa_sLFIPAddr[di] = '' THEN
				diMcNum	:= di - 1;
				EXIT;
			END_IF
		END_FOR

	END_IF

	Act_Background_OPCUA;
	Act_Background_Process;
	Act_Background_Disconnect;

END_ACTION
```

#### Act_Background_OPCUA.st - Do Not Change!!!
```iecst
(** 2020-08-06 **)
ACTION Act_Background_OPCUA:

	IF bRun1 = TRUE THEN

		CASE eOPCUAStep OF

			LFOPCUAStepIncCntr:
				udiNodeCntr	:= udiNodeCntr + 1;

				IF udiNodeCntr > c_diLFClntNum THEN
					udiNodeCntr	:= 1;
				END_IF

				eOPCUAStep	:= LFOPCUAStepChkHdls;

			LFOPCUAStepChkHdls:
				IF pa_sLFIPAddr[udiNodeCntr] <> '' THEN
					IF pa_bLFOnline[udiNodeCntr] = TRUE THEN
						IF a_dwConnectionHdl[udiNodeCntr] <> 0 THEN
							IF a_bNodeWr[udiNodeCntr] = TRUE THEN
								IF a_bNodeRd[udiNodeCntr] = TRUE THEN
									eOPCUAStep	:= LFOPCUAStepWrite;
								ELSE
									eOPCUAStep	:= LFOPCUAStepReadHdls;
								END_IF
							ELSE
								eOPCUAStep	:= LFOPCUAStepWriteHdls;
							END_IF
						ELSE
							eOPCUAStep	:= LFOPCUAStepConnect;
						END_IF
					ELSE
						eOPCUAStep	:= LFOPCUAStepIncCntr;
					END_IF
				ELSE
					udiNodeCntr	:= 0;
					eOPCUAStep	:= LFOPCUAStepStopChk;
				END_IF

			LFOPCUAStepConnect:
				fbConnect.tyOPCUAParam.sIPAddr	:= pa_sLFIPAddr[udiNodeCntr];
				fbConnect(bEn := TRUE);

				IF fbConnect.udiStatus = 0 THEN
					a_dwConnectionHdl[udiNodeCntr]	:= fbConnect.dwConnectionHdl;
					fbConnect(bEn := FALSE);
					eOPCUAStep	:= LFOPCUAStepWriteHdls;
				ELSIF fbConnect.udiStatus < 65534 THEN
					a_dwConnectionHdl[udiNodeCntr]	:= 0;
					fbConnect(bEn := FALSE);
					eOPCUAStep	:= LFOPCUAStepStopChk;
				END_IF

			LFOPCUAStepWriteHdls:
				fbGetNodeHdlListWr.dwConnectionHdl	:= a_dwConnectionHdl[udiNodeCntr];
				fbGetNodeHdlListWr(bEn := TRUE);

				IF fbGetNodeHdlListWr.udiStatus = 0 THEN
					a_bNodeWr[udiNodeCntr]				:= TRUE;
					a_tyWriteHdls[udiNodeCntr].a_dwHdls	:= fbGetNodeHdlListWr.a_dwNodeHdlList;
					fbGetNodeHdlListWr(bEn := FALSE);
					eOPCUAStep	:= LFOPCUAStepReadHdls;
				ELSIF fbGetNodeHdlListWr.udiStatus < 65534 THEN
					a_bNodeWr[udiNodeCntr]	:= FALSE;
					fbGetNodeHdlListWr(bEn := FALSE);
					eOPCUAStep	:= LFOPCUAStepStopChk;
				END_IF

			LFOPCUAStepReadHdls:
				fbGetNodeHdlListRd.dwConnectionHdl	:= a_dwConnectionHdl[udiNodeCntr];
				fbGetNodeHdlListRd(bEn := TRUE);

				IF fbGetNodeHdlListRd.udiStatus = 0 THEN
					a_bNodeRd[udiNodeCntr]				:= TRUE;
					a_tyReadHdls[udiNodeCntr].a_dwHdls	:= fbGetNodeHdlListRd.a_dwNodeHdlList;
					fbGetNodeHdlListRd(bEn := FALSE);
					eOPCUAStep	:= LFOPCUAStepWrite;
				ELSIF fbGetNodeHdlListRd.udiStatus < 65534 THEN
					a_bNodeRd[udiNodeCntr]	:= FALSE;
					fbGetNodeHdlListRd(bEn := FALSE);
					eOPCUAStep	:= LFOPCUAStepStopChk;
				END_IF

			LFOPCUAStepWrite:
				fbWriteList.dwConnectionHdl		:= a_dwConnectionHdl[udiNodeCntr];
				fbWriteList.a_dwNodeHdlList		:= a_tyWriteHdls[udiNodeCntr].a_dwHdls;
				sNodeCntr						:= UDINT_TO_STRING(udiNodeCntr);
				fbWriteList.a_sClientTagNm[0]	:= CONCAT(CONCAT(CONCAT(CONCAT('::' , p_sLeaderProgTagNm) , ':a_tyLeaderToFollowerTag[') , sNodeCntr) , '].sReqProdRcpNm');
				fbWriteList.a_sClientTagNm[1]	:= CONCAT(CONCAT(CONCAT(CONCAT('::' , p_sLeaderProgTagNm) , ':a_tyLeaderToFollowerTag[') , sNodeCntr) , '].diReqProdRcpWidth');
				fbWriteList.a_sClientTagNm[2]	:= CONCAT(CONCAT(CONCAT(CONCAT('::' , p_sLeaderProgTagNm) , ':a_tyLeaderToFollowerTag[') , sNodeCntr) , '].sReqMagRcpNm');
				fbWriteList.a_sClientTagNm[3]	:= CONCAT(CONCAT(CONCAT(CONCAT('::' , p_sLeaderProgTagNm) , ':a_tyLeaderToFollowerTag[') , sNodeCntr) , '].bMnlAccData');
				fbWriteList.a_sClientTagNm[4]	:= CONCAT(CONCAT(CONCAT(CONCAT('::' , p_sLeaderProgTagNm) , ':a_tyLeaderToFollowerTag[') , sNodeCntr) , '].bBypassMnlAccData');
				fbWriteList.a_sClientTagNm[5]	:= CONCAT(CONCAT(CONCAT(CONCAT('::' , p_sLeaderProgTagNm) , ':a_tyLeaderToFollowerTag[') , sNodeCntr) , '].bBlkDS');
				fbWriteList.a_sClientTagNm[6]	:= CONCAT(CONCAT(CONCAT(CONCAT('::' , p_sLeaderProgTagNm) , ':a_tyLeaderToFollowerTag[') , sNodeCntr) , '].bBlkUS');
				fbWriteList.a_sClientTagNm[7]	:= CONCAT(CONCAT(CONCAT(CONCAT('::' , p_sLeaderProgTagNm) , ':a_tyLeaderToFollowerTag[') , sNodeCntr) , '].bSetTm');
				fbWriteList.a_sClientTagNm[8]	:= CONCAT(CONCAT(CONCAT(CONCAT('::' , p_sLeaderProgTagNm) , ':a_tyLeaderToFollowerTag[') , sNodeCntr) , '].dtTm');
				fbWriteList.a_sClientTagNm[9]	:= CONCAT(CONCAT(CONCAT(CONCAT('::' , p_sLeaderProgTagNm) , ':a_tyLeaderToFollowerTag[') , sNodeCntr) , '].uiTmZone');
				fbWriteList.a_sClientTagNm[10]	:= CONCAT(CONCAT(CONCAT(CONCAT('::' , p_sLeaderProgTagNm) , ':a_tyLeaderToFollowerTag[') , sNodeCntr) , '].bBypassWidthChk');
				fbWriteList.a_sClientTagNm[11]	:= CONCAT(CONCAT(CONCAT(CONCAT('::' , p_sLeaderProgTagNm) , ':a_tyLeaderToFollowerTag[') , sNodeCntr) , '].usiRunTm');
				fbWriteList.a_sClientTagNm[12]	:= CONCAT(CONCAT(CONCAT(CONCAT('::' , p_sLeaderProgTagNm) , ':a_tyLeaderToFollowerTag[') , sNodeCntr) , '].bProdNameUSWarn');
				fbWriteList.a_sClientTagNm[13]	:= CONCAT(CONCAT(CONCAT(CONCAT('::' , p_sLeaderProgTagNm) , ':a_tyLeaderToFollowerTag[') , sNodeCntr) , '].bProdNameDSWarn');
				fbWriteList.a_sClientTagNm[14]	:= CONCAT(CONCAT(CONCAT(CONCAT('::' , p_sLeaderProgTagNm) , ':a_tyLeaderToFollowerTag[') , sNodeCntr) , '].bProdWidthUSWarn');
				fbWriteList.a_sClientTagNm[15]	:= CONCAT(CONCAT(CONCAT(CONCAT('::' , p_sLeaderProgTagNm) , ':a_tyLeaderToFollowerTag[') , sNodeCntr) , '].bProdWidthDSWarn');
				fbWriteList.a_sClientTagNm[16]	:= CONCAT(CONCAT(CONCAT(CONCAT('::' , p_sLeaderProgTagNm) , ':a_tyLeaderToFollowerTag[') , sNodeCntr) , '].bLeaderSeqCtrlInActive');
				fbWriteList(bEn := TRUE);

				IF fbWriteList.udiStatus = 0 THEN
					fbWriteList(bEn := FALSE);
					eOPCUAStep	:= LFOPCUAStepRead;
				ELSIF fbWriteList.udiStatus < 65534 THEN
					fbWriteList(bEn := FALSE);
					eOPCUAStep	:= LFOPCUAStepStopChk;
				END_IF

			LFOPCUAStepRead:
				fbReadList.dwConnectionHdl		:= a_dwConnectionHdl[udiNodeCntr];
				fbReadList.a_dwNodeHdlList		:= a_tyReadHdls[udiNodeCntr].a_dwHdls;
				sNodeCntr						:= UDINT_TO_STRING(udiNodeCntr);
				fbReadList.a_sClientTagNm[0]	:= CONCAT(CONCAT(CONCAT(CONCAT('::' , p_sLeaderProgTagNm) , ':a_tyFollowerToLeaderTag[') , sNodeCntr) , '].sCurrProdRcp');
				fbReadList.a_sClientTagNm[1]	:= CONCAT(CONCAT(CONCAT(CONCAT('::' , p_sLeaderProgTagNm) , ':a_tyFollowerToLeaderTag[') , sNodeCntr) , '].diCurrProdWidthUS');
				fbReadList.a_sClientTagNm[2]	:= CONCAT(CONCAT(CONCAT(CONCAT('::' , p_sLeaderProgTagNm) , ':a_tyFollowerToLeaderTag[') , sNodeCntr) , '].sCurrMagRcp');
				fbReadList.a_sClientTagNm[3]	:= CONCAT(CONCAT(CONCAT(CONCAT('::' , p_sLeaderProgTagNm) , ':a_tyFollowerToLeaderTag[') , sNodeCntr) , '].sIPAddr');
				fbReadList.a_sClientTagNm[4]	:= CONCAT(CONCAT(CONCAT(CONCAT('::' , p_sLeaderProgTagNm) , ':a_tyFollowerToLeaderTag[') , sNodeCntr) , '].sMcNm');
				fbReadList.a_sClientTagNm[5]	:= CONCAT(CONCAT(CONCAT(CONCAT('::' , p_sLeaderProgTagNm) , ':a_tyFollowerToLeaderTag[') , sNodeCntr) , '].bSectionLeader');
				fbReadList.a_sClientTagNm[6]	:= CONCAT(CONCAT(CONCAT(CONCAT('::' , p_sLeaderProgTagNm) , ':a_tyFollowerToLeaderTag[') , sNodeCntr) , '].usiRunTm');
				fbReadList.a_sClientTagNm[7]	:= CONCAT(CONCAT(CONCAT(CONCAT('::' , p_sLeaderProgTagNm) , ':a_tyFollowerToLeaderTag[') , sNodeCntr) , '].bProdRcpErr');
				fbReadList.a_sClientTagNm[8]	:= CONCAT(CONCAT(CONCAT(CONCAT('::' , p_sLeaderProgTagNm) , ':a_tyFollowerToLeaderTag[') , sNodeCntr) , '].bProdWidthErr');
				fbReadList.a_sClientTagNm[9]	:= CONCAT(CONCAT(CONCAT(CONCAT('::' , p_sLeaderProgTagNm) , ':a_tyFollowerToLeaderTag[') , sNodeCntr) , '].bMagRcpErr');
				fbReadList.a_sClientTagNm[10]	:= CONCAT(CONCAT(CONCAT(CONCAT('::' , p_sLeaderProgTagNm) , ':a_tyFollowerToLeaderTag[') , sNodeCntr) , '].bSyncTmErr');
				fbReadList.a_sClientTagNm[11]	:= CONCAT(CONCAT(CONCAT(CONCAT('::' , p_sLeaderProgTagNm) , ':a_tyFollowerToLeaderTag[') , sNodeCntr) , '].diCurrProdWidthDS');
				fbReadList.a_sClientTagNm[12]	:= CONCAT(CONCAT(CONCAT(CONCAT('::' , p_sLeaderProgTagNm) , ':a_tyFollowerToLeaderTag[') , sNodeCntr) , '].eCurrMachineStat');
				fbReadList.a_sClientTagNm[13]	:= CONCAT(CONCAT(CONCAT(CONCAT('::' , p_sLeaderProgTagNm) , ':a_tyFollowerToLeaderTag[') , sNodeCntr) , '].bProdChgOverActive');
				fbReadList(bEn := TRUE);

				IF fbReadList.udiStatus = 0 THEN
					fbReadList(bEn := FALSE);
					eOPCUAStep	:= LFOPCUAStepStopChk;
				ELSIF fbReadList.udiStatus < 65534 THEN
					fbReadList(bEn := FALSE);
					eOPCUAStep	:= LFOPCUAStepStopChk;
				END_IF

			LFOPCUAStepStopChk:
				IF bStop AND bStop2Done THEN
					IF bCntr = FALSE THEN
						bCntr	:= TRUE;
					ELSE
						bStop1Done	:= TRUE;
						bCntr		:= FALSE;
					END_IF
				ELSE
					bCntr	:= FALSE;
				END_IF

				eOPCUAStep	:= LFOPCUAStepIncCntr;

		END_CASE

	END_IF

END_ACTION
```

#### Act_Background_Process.st - Do Not Change!!!
```iecst
(** 2020-10-05 **)
ACTION Act_Background_Process:

	IF bRun2 = TRUE AND bStop = FALSE THEN
		fbOnlineChk.a_bOnline				:= pa_bLFOnline;
		fbOnlineChk.a_tyFollowerToLeaderTag	:= a_tyFollowerToLeaderTag;
		fbOnlineChk.diMcNum					:= diMcNum;
		fbOnlineChk(bEn := TRUE);

		fbBlkUSDS.a_tyFollowerToLeaderTag	:= a_tyFollowerToLeaderTag;
		fbBlkUSDS.diBeforeOven1			:= p_diBeforeOven;
		fbBlkUSDS.diAfterOven1			:= p_diAfterOven;
		fbBlkUSDS.diBeforeOven2			:= p_diBeforeOven2;
		fbBlkUSDS.diAfterOven2			:= p_diAfterOven2;
		fbBlkUSDS.diMcNum				:= diMcNum;
		fbBlkUSDS.pa_bLFOnline			:= pa_bLFOnline;
		fbBlkUSDS.bSeqMode				:= (eStat= LFActChgSeqAuto) OR (eStat= LFActChgSeqMnl);
		fbBlkUSDS(bEn := TRUE);

		fbDataUpdt.a_bOnline			:= pa_bLFOnline;
		fbDataUpdt.diMcNum				:= diMcNum;
		fbDataUpdt(bEn := TRUE);

	ELSIF bStop = TRUE THEN
		fbOnlineChk(bEn := FALSE);
		fbBlkUSDS(bEn := FALSE);
		fbDataUpdt(bEn := FALSE);
		bStop2Done	:= TRUE;

	END_IF

END_ACTION
```

#### Act_Background_Disconnect.st - Do Not Change!!!
```iecst
(** 2019-05-07 **)
ACTION Act_Background_Disconnect:

	IF (memcmp(ADR(pa_sLFIPAddr) , ADR(a_sLFIPAddrOld) , SIZEOF(a_sLFIPAddrOld)) <> 0) AND (bDisconnecting = FALSE) THEN
		FOR di := 1 TO c_diLFClntNum DO

			IF pa_sLFIPAddr[di] <> a_sLFIPAddrOld[di] THEN
				diDisconnectIdx	:= di;
				bDisconnecting	:= TRUE;
				EXIT;
			END_IF

		END_FOR
	END_IF

	IF bDisconnecting = TRUE THEN

		IF a_dwConnectionHdl[diDisconnectIdx] <> 0 THEN
			fbDisconnect.dwConnectionHdl	:= a_dwConnectionHdl[diDisconnectIdx];
			fbDisconnect(bEn := TRUE);

			IF fbDisconnect.udiStatus = 0 THEN
				a_dwConnectionHdl[diDisconnectIdx]	:= 0;
				a_bNodeWr[diDisconnectIdx]			:= FALSE;
				a_bNodeRd[diDisconnectIdx]			:= FALSE;
				memset(ADR(a_tyFollowerToLeaderTag[diDisconnectIdx]) , 0 , SIZEOF(a_tyFollowerToLeaderTag[diDisconnectIdx]));
				fbDisconnect(bEn := FALSE);

				a_sLFIPAddrOld[diDisconnectIdx]	:= pa_sLFIPAddr[diDisconnectIdx];
				bDisconnecting						:= FALSE;

			ELSIF fbDisconnect.udiStatus < 65534 THEN
				a_dwConnectionHdl[diDisconnectIdx]	:= 0;
				a_bNodeWr[diDisconnectIdx]			:= FALSE;
				a_bNodeRd[diDisconnectIdx]			:= FALSE;
				memset(ADR(a_tyFollowerToLeaderTag[diDisconnectIdx]) , 0 , SIZEOF(a_tyFollowerToLeaderTag[diDisconnectIdx]));
				fbDisconnect(bEn := FALSE);

				a_sLFIPAddrOld[diDisconnectIdx]	:= pa_sLFIPAddr[diDisconnectIdx];
				bDisconnecting						:= FALSE;

			END_IF

		ELSE
			a_bNodeWr[diDisconnectIdx]	:= FALSE;
			a_bNodeRd[diDisconnectIdx]	:= FALSE;
			memset(ADR(a_tyFollowerToLeaderTag[diDisconnectIdx]) , 0 , SIZEOF(a_tyFollowerToLeaderTag[diDisconnectIdx]));

			a_sLFIPAddrOld[diDisconnectIdx]	:= pa_sLFIPAddr[diDisconnectIdx];
			bDisconnecting						:= FALSE;

		END_IF

	END_IF

END_ACTION
```

#### Act_Main_Disable.st - Do Not Change!!!
```iecst
(** 2019-04-23 **)
ACTION Act_Main_Disable:

END_ACTION
```

#### Act_Alarm.st - Do Not Change!!!
```iecst
(** 2019-04-23 **)
ACTION Act_Alarm:

	//Error
	IF EDGEPOS(eStatus = Error) THEN

		tyAlmData.sProgNm		:= p_sProgNm;
		tyAlmData.udiCode		:= udiStatus;
		tyAlmData.eSeverity		:= AlmSeverityError;
		tyAlmData.udiRunTime	:= tyAlmData.udiRunTime + 1;
		tyAlmData.bAlm			:= TRUE;
		tyAlmData.udiModuleNum  := udiModuleNum;
		g_sLFLeaderProgNm		:= p_sProgNm;
		//Get Error Message
		IF tyAlmData.udiCode < 10000 OR tyAlmData.udiCode > 10099 THEN
			tyAlmData.sAlmMsg	:= 'Unknown';
			tyAlmData.sRcyMsg	:= 'Unknown';
		ELSE
			tyAlmData.sAlmMsg	:= a_tyAlmText[tyAlmData.udiCode].sAlmText;
			tyAlmData.sRcyMsg	:= a_tyAlmText[tyAlmData.udiCode].sRcyText;
		END_IF

		sStatTxt	:= tyAlmData.sAlmMsg;

	ELSIF bRstErr AND (tyAlmData.udiCode <> 0) THEN

		tyAlmData.udiCode	:= 0;
		tyAlmData.eSeverity	:= AlmSeverityNA;
		tyAlmData.sAlmMsg	:= '';
		tyAlmData.sRcyMsg	:= '';
		tyAlmData.bAlm			:= FALSE;
		sStatTxt	:= a_sStatText[eStat];

	END_IF

END_ACTION
```

#### InputRef.var - Do Not Change!!!
```iecst
(*2020-08-06*)
(**)
(*General*)
VAR
	p_eAct : REFERENCE TO eLFAction;
	p_udiRstErr : REFERENCE TO UDINT;
	p_bPrep : REFERENCE TO BOOL;
	p_bEn : REFERENCE TO BOOL;
	p_bDis : REFERENCE TO BOOL;
END_VAR
(**)
(*Input*)
VAR
	p_sReqProdRcpNm : REFERENCE TO STRING[254];
	p_diReqProdWidth : REFERENCE TO DINT;
	p_sReqMagRcpNm : REFERENCE TO STRING[15];
	p_diBeforeOven : REFERENCE TO DINT;
	p_bWidth2Prep : REFERENCE TO BOOL;
	p_diAfterOven : REFERENCE TO DINT;
	p_diBeforeOven2 : REFERENCE TO DINT;
	p_diAfterOven2 : REFERENCE TO DINT;
	p_tOnlineChkDlyTm : REFERENCE TO TIME;
	p_tSetTmOffDlyTm : REFERENCE TO TIME;
	p_dtCurrDT : REFERENCE TO DATE_AND_TIME;
	pa_sLFIPAddr : REFERENCE TO ARRAY[1..c_diLFClntNum] OF STRING[15];
	pa_bLFOnline : REFERENCE TO ARRAY[1..c_diLFClntNum] OF BOOL;
	p_sLeaderProgTagNm : REFERENCE TO STRING[15];
	p_sFollowerProgTagNm : REFERENCE TO STRING[15];
	p_sProgNm : REFERENCE TO STRING[15];
	p_bLFSeqStayActive : REFERENCE TO BOOL;
	p_bNtSettingsLoadDone : REFERENCE TO BOOL;
END_VAR
```

#### Local.var - Do Not Change!!!
```iecst
(*2020-10-05*)
(**)
(*Local Action, State & Status*)
VAR
	eAct : eLFAction := LFActIdle;
	eStat : eLFAction := LFActIdle;
	eStatus : eFBStatus := Idle;
	udiStatus : UDINT := 0;
	sStatTxt : STRING[200] := '';
	a_sStatText : ARRAY[0..50] OF STRING[200] := ['Idling','Background Starting Operations','Background Stopping Operations','Synchronizing PLC Time','Changing All Recipe Automatically','Changing All Recipe Manually','Changing Recipe In Sequence Automatically','Changing Recipe In Sequence Manually',43('')];
END_VAR
(**)
(*Local Alarm*)
VAR
	tyAlmData : tyAlmDat;
	a_tyAlmText : ARRAY[10000..10099] OF tyAlmTxt := [(sAlmText:='Background Not Running While Calling Sync PLC Tm',sRcyText:='Start Background Operations First'),(sAlmText:='Background Not Running While Changing All Recipe Automatically',sRcyText:='Start Background Operations First'),(sAlmText:='Background Not Running While Changing All Recipe Manually',sRcyText:='Start Background Operations First'),(sAlmText:='Background Not Running While Changing Recipe In Sequence Automatically',sRcyText:='Start Background Operations First'),(sAlmText:='Background Not Running While Changing Recipe In Sequence Manually',sRcyText:='Start Background Operations First'),0,94((0))];
END_VAR
(**)
(*Local Output*)
VAR
	a_tyFollowerInfo : ARRAY[1..c_diLFClntNum] OF tyLFFollowerInfo;
	a_tyFollowerToLeaderTag : ARRAY[1..c_diLFClntNum] OF tyLFFollowerToLeaderTag;
END_VAR
(**)
(*Local Input*)
VAR
	udiRstErr : UDINT := 0;
	bPrep : BOOL := TRUE;
	bEn : BOOL := TRUE;
	bDis : BOOL := FALSE;
	sReqProdRcpNm : STRING[254];
	diReqProdWidth : DINT;
	sReqMagRcpNm : STRING[15];
	diBeforeOven : DINT;
	diAfterOven : DINT;
	diBeforeOven2 : DINT;
	diAfterOven2 : DINT;
	bWidth2Prep : BOOL;
	tOnlineChkDlyTm : TIME;
	tSetTmOffDlyTm : TIME;
	dtCurrDT : DATE_AND_TIME;
	a_sLFIPAddr : ARRAY[1..c_diLFClntNum] OF STRING[15];
	a_bLFOnline : ARRAY[1..c_diLFClntNum] OF BOOL;
	sLeaderProgTagNm : STRING[15] := 'LFLeader';
	sFollowerProgTagNm : STRING[15] := 'LFFollower';
	sProgNm : STRING[15] := 'Leader';
	bNtSettingsLoadDone : BOOL := TRUE;
END_VAR
(**)
(*Local*)
VAR
	bRstErr : BOOL;
	udiRstErrOld : UDINT;
	bInitDone : BOOL;
	bInitialDone : BOOL;
	bRun1 : BOOL;
	bRun2 : BOOL;
	bStop : BOOL;
	bStop1Done : BOOL;
	bStop2Done : BOOL;
	bCntr : BOOL;
	di : DINT;
	diDisconnectIdx : DINT := 1;
	diMcNum : DINT;
	a_sLFIPAddrOld : ARRAY[1..c_diLFClntNum] OF STRING[15];
	bDisconnecting : BOOL;
	eStatOld : eLFAction := LFActIdle;
	a_tyLeaderToFollowerTag : ARRAY[1..c_diLFClntNum] OF tyLFLeaderToFollowerTag;
	fbOnlineChk : fbLFLeaderOnlineChk;
	fbSyncTm : fbLFLeaderSyncTm;
	fbChgAll : fbLFLeaderChgAll;
	fbChgSeq : fbLFLeaderChgSeq;
	fbBlkUSDS : fbLFLeaderBlkUSDS;
	fbDataUpdt : fbLFLeaderDataUpdt;
	udiNodeCntr : UDINT;
	sNodeCntr : STRING[80];
	a_dwConnectionHdl : ARRAY[1..c_diLFClntNum] OF DWORD;
	a_bNodeWr : ARRAY[1..c_diLFClntNum] OF BOOL;
	a_bNodeRd : ARRAY[1..c_diLFClntNum] OF BOOL;
	a_tyWriteHdls : ARRAY[1..c_diLFClntNum] OF tyOPCUAHdlList;
	a_tyReadHdls : ARRAY[1..c_diLFClntNum] OF tyOPCUAHdlList;
	eOPCUAStep : eLFOPCUAStep;
	fbConnect : fbOPCUAConnect;
	fbGetNodeHdlListWr : fbOPCUAGetNodeHdlList;
	fbGetNodeHdlListRd : fbOPCUAGetNodeHdlList;
	fbWriteList : fbOPCUAWriteList;
	fbDisconnect : fbOPCUADisconnect;
	fbReadList : fbOPCUAReadList;
	udiModuleNum : UDINT := 3801;
END_VAR
```

### LFFollower.var - Change By Project
```iecst
(*2020-08-06*)
(**)
(*Action & State & Status*)
VAR
	p_LFFollowerStatus : UDINT;
END_VAR
(**)
(*Alarm*)
VAR
	p_LFFollowerAlmData : UDINT;
	p_LFFollowerInfoData : UDINT;
	p_LFFollowerInfoData1 : UDINT;
END_VAR
(**)
(*Output*)
VAR
	p_LFFollowerUSAllow : UDINT;
	p_LFFollowerDSAllow : UDINT;
	p_LFFollowerProdAccDataMnl : UDINT;
	p_LFFollowerProdUpdtDataMnl : UDINT;
	p_LFFollowerMagAccDataMnl : UDINT;
	p_LFFollowerTimeAct : UDINT;
	p_LFFollowerSetDT : UDINT;
	p_LFFollowerWaitRlsBrd : UDINT;
	p_LFFollowerUpdtProdRcp : UDINT;
	p_LFFollowerLdrSeqCtrlInActive : UDINT;
END_VAR
```

### Program Logical/LF/LFFollower (IEC) - 1.00.0 - NtHermes v5.00.0 , NtTCP v5.00.0 , NtMessage v5.00.0

#### InputRef.var
```iecst
(*2021-05-18*)
(**)
(*General*)
VAR
	p_udiRstErr : REFERENCE TO UDINT;
	p_bPrep : REFERENCE TO BOOL;
	p_bEn : REFERENCE TO BOOL;
	p_bDis : REFERENCE TO BOOL;
END_VAR
(**)
(*Configuration*)
VAR
	p_eAWStat : REFERENCE TO eAWAction;
	p_sIPAddr : REFERENCE TO STRING[15];
END_VAR
(**)
(*Input*)
VAR
	p_sMcNm : REFERENCE TO STRING[30];
	p_bAWPrep : REFERENCE TO BOOL;
	p_bAWDis : REFERENCE TO BOOL;
	p_bMnlAccData : REFERENCE TO BOOL;
	p_bSectionLeader : REFERENCE TO BOOL;
	p_sMagRcpNm : REFERENCE TO STRING[30];
	p_diWidthLimit : REFERENCE TO DINT;
	p_bWidth2Prep : REFERENCE TO BOOL;
	p_bUSWidthChkPrep : REFERENCE TO BOOL;
	p_bUSWidthChkEn : REFERENCE TO BOOL;
	p_bUSWidthChkSen : REFERENCE TO BOOL;
	p_bDSWidthChkPrep : REFERENCE TO BOOL;
	p_bDSWidthChkEn : REFERENCE TO BOOL;
	p_bDSWidthChkSen : REFERENCE TO BOOL;
	p_bProdWidthChk : REFERENCE TO BOOL;
	p_bUIProdAccData : REFERENCE TO BOOL;
	p_bUIProdUpdtData : REFERENCE TO BOOL;
	p_bUIMagAccData : REFERENCE TO BOOL;
	p_bDBAOnWOAlign : REFERENCE TO BOOL;
	pa_tyProdRcpList : REFERENCE TO ARRAY[1..c_udiProdRcpMax] OF tyProdRcpParam;
	p_tyCurrProdRcp : REFERENCE TO tyProdRcpParam;
	p_tyDispProdRcp : REFERENCE TO tyProdRcpParam;
	p_sCurrMagRcpNm : REFERENCE TO STRING[30];
	p_eTimeStat : REFERENCE TO eTimeAction;
	p_eTimeStatus : REFERENCE TO eFBStatus;
	p_bAccNewRcpCond : REFERENCE TO BOOL;
	p_bUpdtNewRcpCond : REFERENCE TO BOOL;
	p_bAutoUpdtData : REFERENCE TO BOOL;
	p_sInfoMsg : REFERENCE TO STRING[200];
	p_bInternalUse : REFERENCE TO BOOL;
	p_tyInternalReqProdRcp : REFERENCE TO tyProdRcpParam;
	p_bNewBrdEnteredCond : REFERENCE TO BOOL;
	p_bOldBrdExitedCond : REFERENCE TO BOOL;
	p_bRlsBrd : REFERENCE TO BOOL;
	p_tyToLeaderProdRcp : REFERENCE TO tyProdRcpParam;
	p_bInternalReqProdRcpDiff : REFERENCE TO BOOL;
	p_bUpdtProdRcpDiff : REFERENCE TO BOOL;
	p_bRlsBrdProdRcpDiff : REFERENCE TO BOOL;
	p_sProgNm : REFERENCE TO STRING[15];
	p_bNtSettingsLoadDone : REFERENCE TO BOOL;
	p_tOnlineChkDlyTm : REFERENCE TO TIME;
	p_bManual : REFERENCE TO BOOL;
	p_bErr : REFERENCE TO BOOL;
	p_bWarning : REFERENCE TO BOOL;
	p_bOps : REFERENCE TO BOOL;
	p_bStandby : REFERENCE TO BOOL;
END_VAR
```

#### InputRef_Link.var
```iecst
(*2019-05-07*)
(**)
VAR
	p_bLinkStartupRun : REFERENCE TO BOOL;
	p_eLinkMcParamUSCommMod : REFERENCE TO eMcSetCommMod;
END_VAR
(**)
VAR
	p_bLinkOpsRun : REFERENCE TO BOOL;
	p_bLinkConvHvBrd : REFERENCE TO BOOL;
END_VAR
(**)
VAR
	sWidthInUMTemp : STRING[80];
	p_bLinkUSWidthChkSen : REFERENCE TO BOOL;
	p_bLinkUSWidthChkSen1 : REFERENCE TO BOOL;
	p_bLinkDIInvertHomeSen : REFERENCE TO BOOL;
	p_bLinkDIInvertRemoteSen : REFERENCE TO BOOL;
END_VAR
(**)
VAR
	p_eLinkUIProdRcpAct : REFERENCE TO eProdRcpAction;
	p_eProdRcpStat : REFERENCE TO eProdRcpAction;
	p_eProdRcpStatus : REFERENCE TO eFBStatus;
	p_tyProdRcpCurrRcpWr : REFERENCE TO tyProdRcpParam;
END_VAR
```
